         IF $IN[1896] AND NOT $IN[2172] AND $IN[2171] AND $OUT[4039] OR $TIMER_FLAG[8] THEN
            PREVSTEP = $APP_INT[5]
            $APP_INT[5] = 181
         ENDIF
      ;ENDFOLD
   ;ENDFOLD
   ;FOLD SCHRITT 181 --MS2 Reinigung (an Pneum. Schwenkeinheit MS2)-- ;%{P}%MKUKATPVW,%CSTEP,%VST_NR,%P 1:SCHRITT, 2:181, 3:MS2 Reinigung (an Pneum. Schwenkeinheit MS2)
      ;FOLD ;%{H}
         Case 181
      ;ENDFOLD
      ;FOLD -- Steuerluft EIN -- ;%{SE}%MKUKATPVW %CVW_COM %VCOMMENT %P 2:-- Steuerluft EIN --, 3: VW_COMMENT
      ;ENDFOLD
      ;FOLD A2169 = A4039 ;%{SE}%MKUKATPVW %CVW_SPS %VBOASG %P 2:A2169 = A4039, 3: BOASG
         $OUT[2169] = $OUT[4039]
      ;ENDFOLD
      ;FOLD -- RSK Fehlerausgabe Schwenkeinheit 2 Ruhestellung -- ;%{SE}%MKUKATPVW %CVW_COM %VCOMMENT %P 2:-- RSK Fehlerausgabe Schwenkeinheit 2 Ruhestellung --, 3: VW_COMMENT
      ;ENDFOLD
      ;FOLD F323 = !E2171 & T8 + F323 ;%{SE}%MKUKATPVW %CVW_SPS %VBOASG %P 2:F323 = !E2171 & T8 + F323, 3: BOASG
         $FLAG[323] = NOT $IN[2171] AND $TIMER_FLAG[8] OR $FLAG[323]
      ;ENDFOLD
      ;FOLD -- RSK Sammelstoerung -- ;%{SE}%MKUKATPVW %CVW_COM %VCOMMENT %P 2:-- RSK Sammelstoerung --, 3: VW_COMMENT
      ;ENDFOLD
      ;FOLD F329 = F323 ;%{SE}%MKUKATPVW %CVW_SPS %VBOASG %P 2:F329 = F323, 3: BOASG
         $FLAG[329] = $FLAG[323]
      ;ENDFOLD
      ;FOLD A2171 = AUS ;%{SE}%MKUKATPVW %CVW_SPS %VBOASG %P 2:A2171 = AUS, 3: BOASG
         $OUT[2171] = FALSE
      ;ENDFOLD
      ;FOLD -- FRG Bewegung AUS -- ;%{SE}%MKUKATPVW %CVW_COM %VCOMMENT %P 2:-- FRG Bewegung AUS --, 3: VW_COMMENT
      ;ENDFOLD
      ;FOLD A2174 = AUS ;%{SE}%MKUKATPVW %CVW_SPS %VBOASG %P 2:A2174 = AUS, 3: BOASG
         $OUT[2174] = FALSE
      ;ENDFOLD
      ;FOLD Schritt 178 = F323 & (E26 + E27) & A4039 ;%{SE}%MKUKATPVW %CVW_SPS %VST_CON %P 2:Schritt 178 = F323 & (E26 + E27) & A4039, 3: ST_CON
         IF $FLAG[323] AND ($IN[26] OR $IN[27]) AND $OUT[4039] THEN
            PREVSTEP = $APP_INT[5]
            $APP_INT[5] = 178
         ENDIF
      ;ENDFOLD
      ;FOLD Schritt 182 = !F323 & E2174 & A4039 ;%{SE}%MKUKATPVW %CVW_SPS %VST_CON %P 2:Schritt 182 = !F323 & E2174 & A4039, 3: ST_CON
         IF NOT $FLAG[323] AND $IN[2174] AND $OUT[4039] THEN
            PREVSTEP = $APP_INT[5]
            $APP_INT[5] = 182
         ENDIF
      ;ENDFOLD
   ;ENDFOLD
   ;FOLD SCHRITT 182 --MS2 Reinigung (an Pneum. Schwenkeinheit MS2)-- ;%{P}%MKUKATPVW,%CSTEP,%VST_NR,%P 1:SCHRITT, 2:182, 3:MS2 Reinigung (an Pneum. Schwenkeinheit MS2)
      ;FOLD ;%{H}
         Case 182
      ;ENDFOLD
      ;FOLD -- Steuerluft EIN -- ;%{SE}%MKUKATPVW %CVW_COM %VCOMMENT %P 2:-- Steuerluft EIN --, 3: VW_COMMENT
      ;ENDFOLD
      ;FOLD A2169 = A4039 ;%{SE}%MKUKATPVW %CVW_SPS %VBOASG %P 2:A2169 = A4039, 3: BOASG
         $OUT[2169] = $OUT[4039]
      ;ENDFOLD
      ;FOLD F329 = T8 ;%{SE}%MKUKATPVW %CVW_SPS %VBOASG %P 2:F329 = T8, 3: BOASG
         $FLAG[329] = $TIMER_FLAG[8]
      ;ENDFOLD
      ;FOLD F323 = AUS ;%{SE}%MKUKATPVW %CVW_SPS %VBOASG %P 2:F323 = AUS, 3: BOASG
         $FLAG[323] = FALSE
      ;ENDFOLD
      ;FOLD -- FRG in Endlage halten ein -- ;%{SE}%MKUKATPVW %CVW_COM %VCOMMENT %P 2:-- FRG in Endlage halten ein --, 3: VW_COMMENT
      ;ENDFOLD
      ;FOLD A2173 = EIN ;%{SE}%MKUKATPVW %CVW_SPS %VBOASG %P 2:A2173 = EIN, 3: BOASG
         $OUT[2173] = TRUE
      ;ENDFOLD
      ;FOLD Schritt 183 = E2173 & A4039 ;%{SE}%MKUKATPVW %CVW_SPS %VST_CON %P 2:Schritt 183 = E2173 & A4039, 3: ST_CON
         IF $IN[2173] AND $OUT[4039] THEN
            PREVSTEP = $APP_INT[5]
            $APP_INT[5] = 183
         ENDIF
      ;ENDFOLD
   ;ENDFOLD
   ;FOLD SCHRITT 183 --MS2 Reinigung (an Pneum. Schwenkeinheit MS2)-- ;%{P}%MKUKATPVW,%CSTEP,%VST_NR,%P 1:SCHRITT, 2:183, 3:MS2 Reinigung (an Pneum. Schwenkeinheit MS2)
      ;FOLD ;%{H}
         Case 183
      ;ENDFOLD
      ;FOLD -- Steuerluft EIN -- ;%{SE}%MKUKATPVW %CVW_COM %VCOMMENT %P 2:-- Steuerluft EIN --, 3: VW_COMMENT
      ;ENDFOLD
      ;FOLD A2169 = A4039 ;%{SE}%MKUKATPVW %CVW_SPS %VBOASG %P 2:A2169 = A4039, 3: BOASG
         $OUT[2169] = $OUT[4039]
      ;ENDFOLD
      ;FOLD -- FRG in Endlage halten AUS -- ;%{SE}%MKUKATPVW %CVW_COM %VCOMMENT %P 2:-- FRG in Endlage halten AUS --, 3: VW_COMMENT
      ;ENDFOLD
      ;FOLD A2173 = AUS ;%{SE}%MKUKATPVW %CVW_SPS %VBOASG %P 2:A2173 = AUS, 3: BOASG
         $OUT[2173] = FALSE
      ;ENDFOLD
      ;FOLD -- MS1 Zaehler ruecksetzen -- ;%{SE}%MKUKATPVW %CVW_COM %VCOMMENT %P 2:-- MS1 Zaehler ruecksetzen --, 3: VW_COMMENT
      ;ENDFOLD
      ;FOLD -- MS1 FRG Reinigung -- ;%{SE}%MKUKATPVW %CVW_COM %VCOMMENT %P 2:-- MS1 FRG Reinigung --, 3: VW_COMMENT
      ;ENDFOLD
      ;FOLD F607 = AUS ;%{SE}%MKUKATPVW %CVW_SPS %VBOASG %P 2:F607 = AUS, 3: BOASG
         $FLAG[607] = FALSE
      ;ENDFOLD
      ;FOLD -- MS1 Reinigung FK -- ;%{SE}%MKUKATPVW %CVW_COM %VCOMMENT %P 2:-- MS1 Reinigung FK --, 3: VW_COMMENT
      ;ENDFOLD
      ;FOLD F609 = EIN ;%{SE}%MKUKATPVW %CVW_SPS %VBOASG %P 2:F609 = EIN, 3: BOASG
         $FLAG[609] = TRUE
      ;ENDFOLD
      ;FOLD t8 ( EIN ) = STOP ;%{SE}%MKUKATPVW %CVW_SPS %VTSTOP %P 2:t8 ( EIN ) = STOP, 3: TSTOP
         VW(#SET_TIME,TRUE,8,1,0)
      ;ENDFOLD
      ;FOLD Schritt 1 = A4039 ;%{SE}%MKUKATPVW %CVW_SPS %VST_CON %P 2:Schritt 1 = A4039, 3: ST_CON
         IF $OUT[4039] THEN
            PREVSTEP = $APP_INT[5]
            $APP_INT[5] = 1
         ENDIF
      ;ENDFOLD
   ;ENDFOLD
   ;FOLD SCHRITT 184 -- Reserviert -- ;%{P}%MKUKATPVW,%CSTEP,%VST_NR,%P 1:SCHRITT, 2:184, 3: Reserviert
      ;FOLD ;%{H}
         Case 184
      ;ENDFOLD
      ;FOLD 1:;%{SE} %MKUKATPVW
      ;ENDFOLD
   ;ENDFOLD
   ;FOLD SCHRITT 185 -- Reserviert -- ;%{P}%MKUKATPVW,%CSTEP,%VST_NR,%P 1:SCHRITT, 2:185, 3: Reserviert
      ;FOLD ;%{H}
         Case 185
      ;ENDFOLD
      ;FOLD 1:;%{SE} %MKUKATPVW
      ;ENDFOLD
   ;ENDFOLD
   ;FOLD SCHRITT 186 -- Reserviert -- ;%{P}%MKUKATPVW,%CSTEP,%VST_NR,%P 1:SCHRITT, 2:186, 3: Reserviert
      ;FOLD ;%{H}
         Case 186
      ;ENDFOLD
      ;FOLD 1:;%{SE} %MKUKATPVW
      ;ENDFOLD
   ;ENDFOLD
   ;FOLD SCHRITT 187 -- Reserviert -- ;%{P}%MKUKATPVW,%CSTEP,%VST_NR,%P 1:SCHRITT, 2:187, 3: Reserviert
      ;FOLD ;%{H}
         Case 187
      ;ENDFOLD
      ;FOLD 1:;%{SE} %MKUKATPVW
      ;ENDFOLD
   ;ENDFOLD
   ;FOLD SCHRITT 188 -- Reserviert -- ;%{P}%MKUKATPVW,%CSTEP,%VST_NR,%P 1:SCHRITT, 2:188, 3: Reserviert
      ;FOLD ;%{H}
         Case 188
      ;ENDFOLD
      ;FOLD 1:;%{SE} %MKUKATPVW
      ;ENDFOLD
   ;ENDFOLD
   ;FOLD SCHRITT 189 -- Reserviert -- ;%{P}%MKUKATPVW,%CSTEP,%VST_NR,%P 1:SCHRITT, 2:189, 3: Reserviert
      ;FOLD ;%{H}
         Case 189
      ;ENDFOLD
      ;FOLD 1:;%{SE} %MKUKATPVW
      ;ENDFOLD
   ;ENDFOLD
   ;FOLD SCHRITT 190 -- Reserviert -- ;%{P}%MKUKATPVW,%CSTEP,%VST_NR,%P 1:SCHRITT, 2:190, 3: Reserviert
      ;FOLD ;%{H}
         Case 190
      ;ENDFOLD
      ;FOLD 1:;%{SE} %MKUKATPVW
      ;ENDFOLD
   ;ENDFOLD
   ;FOLD SCHRITT 191 -- Reserviert -- ;%{P}%MKUKATPVW,%CSTEP,%VST_NR,%P 1:SCHRITT, 2:191, 3: Reserviert
      ;FOLD ;%{H}
         Case 191
      ;ENDFOLD
      ;FOLD 1:;%{SE} %MKUKATPVW
      ;ENDFOLD
   ;ENDFOLD
   ;FOLD SCHRITT 192 -- Reserviert -- ;%{P}%MKUKATPVW,%CSTEP,%VST_NR,%P 1:SCHRITT, 2:192, 3: Reserviert
      ;FOLD ;%{H}
         Case 192
      ;ENDFOLD
      ;FOLD 1:;%{SE} %MKUKATPVW
      ;ENDFOLD
   ;ENDFOLD
   ;FOLD SCHRITT 193 -- Reserviert -- ;%{P}%MKUKATPVW,%CSTEP,%VST_NR,%P 1:SCHRITT, 2:193, 3: Reserviert
      ;FOLD ;%{H}
         Case 193
      ;ENDFOLD
      ;FOLD 1:;%{SE} %MKUKATPVW
      ;ENDFOLD
   ;ENDFOLD
   ;FOLD SCHRITT 194 -- Reserviert -- ;%{P}%MKUKATPVW,%CSTEP,%VST_NR,%P 1:SCHRITT, 2:194, 3: Reserviert
      ;FOLD ;%{H}
         Case 194
      ;ENDFOLD
      ;FOLD 1:;%{SE} %MKUKATPVW
      ;ENDFOLD
   ;ENDFOLD
   ;FOLD SCHRITT 195 -- Reserviert -- ;%{P}%MKUKATPVW,%CSTEP,%VST_NR,%P 1:SCHRITT, 2:195, 3: Reserviert
      ;FOLD ;%{H}
         Case 195
      ;ENDFOLD
      ;FOLD 1:;%{SE} %MKUKATPVW
      ;ENDFOLD
   ;ENDFOLD
   ;FOLD SCHRITT 196 -- Reserviert -- ;%{P}%MKUKATPVW,%CSTEP,%VST_NR,%P 1:SCHRITT, 2:196, 3: Reserviert
      ;FOLD ;%{H}
         Case 196
      ;ENDFOLD
      ;FOLD 1:;%{SE} %MKUKATPVW
      ;ENDFOLD
   ;ENDFOLD
   ;FOLD SCHRITT 197 -- Reserviert -- ;%{P}%MKUKATPVW,%CSTEP,%VST_NR,%P 1:SCHRITT, 2:197, 3: Reserviert
      ;FOLD ;%{H}
         Case 197
      ;ENDFOLD
      ;FOLD 1:;%{SE} %MKUKATPVW
      ;ENDFOLD
   ;ENDFOLD
   ;FOLD SCHRITT 198 -- Reserviert -- ;%{P}%MKUKATPVW,%CSTEP,%VST_NR,%P 1:SCHRITT, 2:198, 3: Reserviert
      ;FOLD ;%{H}
         Case 198
      ;ENDFOLD
      ;FOLD 1:;%{SE} %MKUKATPVW
      ;ENDFOLD
   ;ENDFOLD
   ;FOLD SCHRITT 199 -- Reserviert -- ;%{P}%MKUKATPVW,%CSTEP,%VST_NR,%P 1:SCHRITT, 2:199, 3: Reserviert
      ;FOLD ;%{H}
         Case 199
      ;ENDFOLD
      ;FOLD 1:;%{SE} %MKUKATPVW
      ;ENDFOLD
   ;ENDFOLD
   ;FOLD SCHRITT 200 -- Reserviert -- ;%{P}%MKUKATPVW,%CSTEP,%VST_NR,%P 1:SCHRITT, 2:200, 3: Reserviert
      ;FOLD ;%{H}
         Case 200
      ;ENDFOLD
      ;FOLD 1:;%{SE} %MKUKATPVW
      ;ENDFOLD
   ;ENDFOLD
   ;FOLD SCHRITT 201 -- Reserviert -- ;%{P}%MKUKATPVW,%CSTEP,%VST_NR,%P 1:SCHRITT, 2:201, 3: Reserviert
      ;FOLD ;%{H}
         Case 201
      ;ENDFOLD
      ;FOLD 1:;%{SE} %MKUKATPVW
      ;ENDFOLD
   ;ENDFOLD
   ;FOLD SCHRITT 202 -- Reserviert -- ;%{P}%MKUKATPVW,%CSTEP,%VST_NR,%P 1:SCHRITT, 2:202, 3: Reserviert
      ;FOLD ;%{H}
         Case 202
      ;ENDFOLD
      ;FOLD 1:;%{SE} %MKUKATPVW
      ;ENDFOLD
   ;ENDFOLD
   ;FOLD SCHRITT 203 -- Reserviert -- ;%{P}%MKUKATPVW,%CSTEP,%VST_NR,%P 1:SCHRITT, 2:203, 3: Reserviert
      ;FOLD ;%{H}
         Case 203
      ;ENDFOLD
      ;FOLD 1:;%{SE} %MKUKATPVW
      ;ENDFOLD
   ;ENDFOLD
   ;FOLD SCHRITT 204 -- Reserviert -- ;%{P}%MKUKATPVW,%CSTEP,%VST_NR,%P 1:SCHRITT, 2:204, 3: Reserviert
      ;FOLD ;%{H}
         Case 204
      ;ENDFOLD
      ;FOLD 1:;%{SE} %MKUKATPVW
      ;ENDFOLD
   ;ENDFOLD
   ;FOLD SCHRITT 205 -- Reserviert -- ;%{P}%MKUKATPVW,%CSTEP,%VST_NR,%P 1:SCHRITT, 2:205, 3: Reserviert
      ;FOLD ;%{H}
         Case 205
      ;ENDFOLD
      ;FOLD 1:;%{SE} %MKUKATPVW
      ;ENDFOLD
   ;ENDFOLD
   ;FOLD SCHRITT 206 -- Reserviert -- ;%{P}%MKUKATPVW,%CSTEP,%VST_NR,%P 1:SCHRITT, 2:206, 3: Reserviert
      ;FOLD ;%{H}
         Case 206
      ;ENDFOLD
      ;FOLD 1:;%{SE} %MKUKATPVW
      ;ENDFOLD
   ;ENDFOLD
   ;FOLD SCHRITT 207 -- Reserviert -- ;%{P}%MKUKATPVW,%CSTEP,%VST_NR,%P 1:SCHRITT, 2:207, 3: Reserviert
      ;FOLD ;%{H}
         Case 207
      ;ENDFOLD
      ;FOLD 1:;%{SE} %MKUKATPVW
      ;ENDFOLD
   ;ENDFOLD
   ;FOLD SCHRITT 208 -- Reserviert -- ;%{P}%MKUKATPVW,%CSTEP,%VST_NR,%P 1:SCHRITT, 2:208, 3: Reserviert
      ;FOLD ;%{H}
         Case 208
      ;ENDFOLD
      ;FOLD 1:;%{SE} %MKUKATPVW
      ;ENDFOLD
   ;ENDFOLD
   ;FOLD SCHRITT 209 -- Reserviert -- ;%{P}%MKUKATPVW,%CSTEP,%VST_NR,%P 1:SCHRITT, 2:209, 3: Reserviert
      ;FOLD ;%{H}
         Case 209
      ;ENDFOLD
      ;FOLD 1:;%{SE} %MKUKATPVW
      ;ENDFOLD
   ;ENDFOLD
   ;FOLD SCHRITT 210 -- Reserviert -- ;%{P}%MKUKATPVW,%CSTEP,%VST_NR,%P 1:SCHRITT, 2:210, 3: Reserviert
      ;FOLD ;%{H}
         Case 210
      ;ENDFOLD
      ;FOLD 1:;%{SE} %MKUKATPVW
      ;ENDFOLD
   ;ENDFOLD
   ;FOLD SCHRITT 211 -- Reserviert -- ;%{P}%MKUKATPVW,%CSTEP,%VST_NR,%P 1:SCHRITT, 2:211, 3: Reserviert
      ;FOLD ;%{H}
         Case 211
      ;ENDFOLD
      ;FOLD 1:;%{SE} %MKUKATPVW
      ;ENDFOLD
   ;ENDFOLD
   ;FOLD SCHRITT 212 -- Reserviert -- ;%{P}%MKUKATPVW,%CSTEP,%VST_NR,%P 1:SCHRITT, 2:212, 3: Reserviert
      ;FOLD ;%{H}
         Case 212
      ;ENDFOLD
      ;FOLD 1:;%{SE} %MKUKATPVW
      ;ENDFOLD
   ;ENDFOLD
   ;FOLD SCHRITT 213 -- Reserviert -- ;%{P}%MKUKATPVW,%CSTEP,%VST_NR,%P 1:SCHRITT, 2:213, 3: Reserviert
      ;FOLD ;%{H}
         Case 213
      ;ENDFOLD
      ;FOLD 1:;%{SE} %MKUKATPVW
      ;ENDFOLD
   ;ENDFOLD
   ;FOLD SCHRITT 214 -- Reserviert -- ;%{P}%MKUKATPVW,%CSTEP,%VST_NR,%P 1:SCHRITT, 2:214, 3: Reserviert
      ;FOLD ;%{H}
         Case 214
      ;ENDFOLD
      ;FOLD 1:;%{SE} %MKUKATPVW
      ;ENDFOLD
   ;ENDFOLD
   ;FOLD SCHRITT 215 -- Reserviert -- ;%{P}%MKUKATPVW,%CSTEP,%VST_NR,%P 1:SCHRITT, 2:215, 3: Reserviert
      ;FOLD ;%{H}
         Case 215
      ;ENDFOLD
      ;FOLD 1:;%{SE} %MKUKATPVW
      ;ENDFOLD
   ;ENDFOLD
   ;FOLD SCHRITT 216 -- Reserviert -- ;%{P}%MKUKATPVW,%CSTEP,%VST_NR,%P 1:SCHRITT, 2:216, 3: Reserviert
      ;FOLD ;%{H}
         Case 216
      ;ENDFOLD
      ;FOLD 1:;%{SE} %MKUKATPVW
      ;ENDFOLD
   ;ENDFOLD
   ;FOLD SCHRITT 217 -- STAT EZ1/SP1/KE1 Setzhub 2 -- ;%{P}%MKUKATPVW,%CSTEP,%VST_NR,%P 1:SCHRITT, 2:217, 3: STAT EZ1/SP1/KE1 Setzhub 2
      ;FOLD ;%{H}
         Case 217
      ;ENDFOLD
      ;FOLD -- Druckvorgabe SK1/EZ1/SP1/KE1 -- ;%{SE}%MKUKATPVW %CVW_COM %VCOMMENT %P 2:-- Druckvorgabe SK1/EZ1/SP1/KE1 --, 3: VW_COMMENT
      ;ENDFOLD
      ;FOLD F168 = F78 & !F830 ;%{SE}%MKUKATPVW %CVW_SPS %VBOASG %P 2:F168 = F78 & !F830, 3: BOASG
         $FLAG[168] = $FLAG[78] AND NOT $FLAG[830]
      ;ENDFOLD
      ;FOLD bin1 ( F168 ) = 61 ;%{SE}%MKUKATPVW %CVW_SPS %VARIASG %P 2:bin1 ( F168 ) = 61, 3: ARIASG
         VW(#BINOUT,$FLAG[168],1,61)
      ;ENDFOLD
      ;FOLD F168 = AUS ;%{SE}%MKUKATPVW %CVW_SPS %VBOASG %P 2:F168 = AUS, 3: BOASG
         $FLAG[168] = FALSE
      ;ENDFOLD
      ;FOLD bin3 ( F78 ) = 61 ;%{SE}%MKUKATPVW %CVW_SPS %VARIASG %P 2:bin3 ( F78 ) = 61, 3: ARIASG
         VW(#BINOUT,$FLAG[78],3,61)
      ;ENDFOLD
      ;FOLD -- Wartezeit Programmwechsel SK -- ;%{SE}%MKUKATPVW %CVW_COM %VCOMMENT %P 2:-- Wartezeit Programmwechsel SK --, 3: VW_COMMENT
      ;ENDFOLD
      ;FOLD T8 ( !F334 ) = -2[1/10Sek] ;%{SE}%MKUKATPVW %CVW_SPS %VTASG %P 2:T8 ( !F334 ) = -2[1/10Sek], 3: TASG
         VW(#SET_TIME,NOT $FLAG[334],8,0,-2)
      ;ENDFOLD
      ;FOLD -- Hilfsflag SK Programmwechsel -- ;%{SE}%MKUKATPVW %CVW_COM %VCOMMENT %P 2:-- Hilfsflag SK Programmwechsel --, 3: VW_COMMENT
      ;ENDFOLD
      ;FOLD F334 = EIN ;%{SE}%MKUKATPVW %CVW_SPS %VBOASG %P 2:F334 = EIN, 3: BOASG
         $FLAG[334] = TRUE
      ;ENDFOLD
      ;FOLD Schritt 218 = T8 & A4039 ;%{SE}%MKUKATPVW %CVW_SPS %VST_CON %P 2:Schritt 218 = T8 & A4039, 3: ST_CON
         IF $TIMER_FLAG[8] AND $OUT[4039] THEN
            PREVSTEP = $APP_INT[5]
            $APP_INT[5] = 218
         ENDIF
      ;ENDFOLD
   ;ENDFOLD
   ;FOLD SCHRITT 218 -- STAT EZ1/SP1/KE1 Setzhub 2 -- ;%{P}%MKUKATPVW,%CSTEP,%VST_NR,%P 1:SCHRITT, 2:218, 3: STAT EZ1/SP1/KE1 Setzhub 2
      ;FOLD ;%{H}
         Case 218
      ;ENDFOLD
      ;FOLD -- Hilfsflag SK Programmwechsel -- ;%{SE}%MKUKATPVW %CVW_COM %VCOMMENT %P 2:-- Hilfsflag SK Programmwechsel --, 3: VW_COMMENT
      ;ENDFOLD
      ;FOLD F334 = AUS ;%{SE}%MKUKATPVW %CVW_SPS %VBOASG %P 2:F334 = AUS, 3: BOASG
         $FLAG[334] = FALSE
      ;ENDFOLD
      ;FOLD -- Zeit fuer Setzhub -- ;%{SE}%MKUKATPVW %CVW_COM %VCOMMENT %P 2:-- Zeit fuer Setzhub --, 3: VW_COMMENT
      ;ENDFOLD
      ;FOLD T8 ( EIN ) = -15[1/10Sek] ;%{SE}%MKUKATPVW %CVW_SPS %VTASG %P 2:T8 ( EIN ) = -15[1/10Sek], 3: TASG
         VW(#SET_TIME,TRUE,8,0,-15)
      ;ENDFOLD
      ;FOLD Schritt 219 = A4039 ;%{SE}%MKUKATPVW %CVW_SPS %VST_CON %P 2:Schritt 219 = A4039, 3: ST_CON
         IF $OUT[4039] THEN
            PREVSTEP = $APP_INT[5]
            $APP_INT[5] = 219
         ENDIF
      ;ENDFOLD
   ;ENDFOLD
   ;FOLD SCHRITT 219 -- STAT EZ1/SP1/KE1 Setzhub 2 -- ;%{P}%MKUKATPVW,%CSTEP,%VST_NR,%P 1:SCHRITT, 2:219, 3: STAT EZ1/SP1/KE1 Setzhub 2
      ;FOLD ;%{H}
         Case 219
      ;ENDFOLD
      ;FOLD -- Hilfsflag SK Programmwechsel -- ;%{SE}%MKUKATPVW %CVW_COM %VCOMMENT %P 2:-- Hilfsflag SK Programmwechsel --, 3: VW_COMMENT
      ;ENDFOLD
      ;FOLD F334 = AUS ;%{SE}%MKUKATPVW %CVW_SPS %VBOASG %P 2:F334 = AUS, 3: BOASG
         $FLAG[334] = FALSE
      ;ENDFOLD
      ;FOLD -- EZ1/SP1/KE1 schliessen -- ;%{SE}%MKUKATPVW %CVW_COM %VCOMMENT %P 2:-- EZ1/SP1/KE1 schliessen --, 3: VW_COMMENT
      ;ENDFOLD
      ;FOLD A717 = AUS ;%{SE}%MKUKATPVW %CVW_SPS %VBOASG %P 2:A717 = AUS, 3: BOASG
         $OUT[717] = FALSE
      ;ENDFOLD
      ;FOLD -- EZ1/SP1 -- ;%{SE}%MKUKATPVW %CVW_COM %VCOMMENT %P 2:-- EZ1/SP1 --, 3: VW_COMMENT
      ;ENDFOLD
      ;FOLD A718 = !F329 & !F122 & !F830 ;%{SE}%MKUKATPVW %CVW_SPS %VBOASG %P 2:A718 = !F329 & !F122 & !F830, 3: BOASG
         $OUT[718] = NOT $FLAG[329] AND NOT $FLAG[122] AND NOT $FLAG[830]
      ;ENDFOLD
      ;FOLD -- KE1 -- ;%{SE}%MKUKATPVW %CVW_COM %VCOMMENT %P 2:-- KE1 --, 3: VW_COMMENT
      ;ENDFOLD
      ;FOLD A766 = !F329 & !F122 & F830 ;%{SE}%MKUKATPVW %CVW_SPS %VBOASG %P 2:A766 = !F329 & !F122 & F830, 3: BOASG
         $OUT[766] = NOT $FLAG[329] AND NOT $FLAG[122] AND $FLAG[830]
      ;ENDFOLD
      ;FOLD Schritt 220 = (!E717 & E718 & T8 + T9) & A4039 ;%{SE}%MKUKATPVW %CVW_SPS %VST_CON %P 2:Schritt 220 = (!E717 & E718 & T8 + T9) & A4039, 3: ST_CON
         IF (NOT $IN[717] AND $IN[718] AND $TIMER_FLAG[8] OR $TIMER_FLAG[9]) AND $OUT[4039] THEN
            PREVSTEP = $APP_INT[5]
            $APP_INT[5] = 220
         ENDIF
      ;ENDFOLD
   ;ENDFOLD
   ;FOLD SCHRITT 220 -- STAT EZ1/SP1/KE1 Setzhub 2 -- ;%{P}%MKUKATPVW,%CSTEP,%VST_NR,%P 1:SCHRITT, 2:220, 3: STAT EZ1/SP1/KE1 Setzhub 2
      ;FOLD ;%{H}
         Case 220
      ;ENDFOLD
      ;FOLD -- RSK Fehlerausgabe Kraftaufbau -- ;%{SE}%MKUKATPVW %CVW_COM %VCOMMENT %P 2:-- RSK Fehlerausgabe Kraftaufbau --, 3: VW_COMMENT
      ;ENDFOLD
      ;FOLD F325 = !E718 & T9 ;%{SE}%MKUKATPVW %CVW_SPS %VBOASG %P 2:F325 = !E718 & T9, 3: BOASG
         $FLAG[325] = NOT $IN[718] AND $TIMER_FLAG[9]
      ;ENDFOLD
      ;FOLD F329 = T9 ;%{SE}%MKUKATPVW %CVW_SPS %VBOASG %P 2:F329 = T9, 3: BOASG
         $FLAG[329] = $TIMER_FLAG[9]
      ;ENDFOLD
      ;FOLD -- EZ1/SP1/KE1 SZ1 oeffnen -- ;%{SE}%MKUKATPVW %CVW_COM %VCOMMENT %P 2:-- EZ1/SP1/KE1 SZ1 oeffnen --, 3: VW_COMMENT
      ;ENDFOLD
      ;FOLD A718 = AUS ;%{SE}%MKUKATPVW %CVW_SPS %VBOASG %P 2:A718 = AUS, 3: BOASG
         $OUT[718] = FALSE
      ;ENDFOLD
      ;FOLD A766 = AUS ;%{SE}%MKUKATPVW %CVW_SPS %VBOASG %P 2:A766 = AUS, 3: BOASG
         $OUT[766] = FALSE
      ;ENDFOLD
      ;FOLD A717 = EIN ;%{SE}%MKUKATPVW %CVW_SPS %VBOASG %P 2:A717 = EIN, 3: BOASG
         $OUT[717] = TRUE
      ;ENDFOLD
      ;FOLD -- Druckvorgabe SK1/EZ1/SP1/KE1 -- ;%{SE}%MKUKATPVW %CVW_COM %VCOMMENT %P 2:-- Druckvorgabe SK1/EZ1/SP1/KE1 --, 3: VW_COMMENT
      ;ENDFOLD
      ;FOLD F168 = F78 & !F830 ;%{SE}%MKUKATPVW %CVW_SPS %VBOASG %P 2:F168 = F78 & !F830, 3: BOASG
         $FLAG[168] = $FLAG[78] AND NOT $FLAG[830]
      ;ENDFOLD
      ;FOLD bin1 ( F168 ) = 41 ;%{SE}%MKUKATPVW %CVW_SPS %VARIASG %P 2:bin1 ( F168 ) = 41, 3: ARIASG
         VW(#BINOUT,$FLAG[168],1,41)
      ;ENDFOLD
      ;FOLD F168 = F79 & !F830 ;%{SE}%MKUKATPVW %CVW_SPS %VBOASG %P 2:F168 = F79 & !F830, 3: BOASG
         $FLAG[168] = $FLAG[79] AND NOT $FLAG[830]
      ;ENDFOLD
      ;FOLD bin1 ( F79 ) = 51 ;%{SE}%MKUKATPVW %CVW_SPS %VARIASG %P 2:bin1 ( F79 ) = 51, 3: ARIASG
         VW(#BINOUT,$FLAG[79],1,51)
      ;ENDFOLD
      ;FOLD F168 = AUS ;%{SE}%MKUKATPVW %CVW_SPS %VBOASG %P 2:F168 = AUS, 3: BOASG
         $FLAG[168] = FALSE
      ;ENDFOLD
      ;FOLD bin3 ( F78 ) = 41 ;%{SE}%MKUKATPVW %CVW_SPS %VARIASG %P 2:bin3 ( F78 ) = 41, 3: ARIASG
         VW(#BINOUT,$FLAG[78],3,41)
      ;ENDFOLD
      ;FOLD bin3 ( F79 ) = 51 ;%{SE}%MKUKATPVW %CVW_SPS %VARIASG %P 2:bin3 ( F79 ) = 51, 3: ARIASG
         VW(#BINOUT,$FLAG[79],3,51)
      ;ENDFOLD
      ;FOLD -- Wartezeit Programmwechsel SK -- ;%{SE}%MKUKATPVW %CVW_COM %VCOMMENT %P 2:-- Wartezeit Programmwechsel SK --, 3: VW_COMMENT
      ;ENDFOLD
      ;FOLD T8 ( !F334 ) = -2[1/10Sek] ;%{SE}%MKUKATPVW %CVW_SPS %VTASG %P 2:T8 ( !F334 ) = -2[1/10Sek], 3: TASG
         VW(#SET_TIME,NOT $FLAG[334],8,0,-2)
      ;ENDFOLD
      ;FOLD -- Hilfsflag SK Programmwechsel -- ;%{SE}%MKUKATPVW %CVW_COM %VCOMMENT %P 2:-- Hilfsflag SK Programmwechsel --, 3: VW_COMMENT
      ;ENDFOLD
      ;FOLD F334 = EIN ;%{SE}%MKUKATPVW %CVW_SPS %VBOASG %P 2:F334 = EIN, 3: BOASG
         $FLAG[334] = TRUE
      ;ENDFOLD
      ;FOLD Schritt 221 = T8 & A4039 ;%{SE}%MKUKATPVW %CVW_SPS %VST_CON %P 2:Schritt 221 = T8 & A4039, 3: ST_CON
         IF $TIMER_FLAG[8] AND $OUT[4039] THEN
            PREVSTEP = $APP_INT[5]
            $APP_INT[5] = 221
         ENDIF
      ;ENDFOLD
   ;ENDFOLD
   ;FOLD SCHRITT 221 -- STAT EZ1/SP1/KE1 Setzhub 2 -- ;%{P}%MKUKATPVW,%CSTEP,%VST_NR,%P 1:SCHRITT, 2:221, 3: STAT EZ1/SP1/KE1 Setzhub 2
      ;FOLD ;%{H}
         Case 221
      ;ENDFOLD
      ;FOLD -- Hilfsflag SK Programmwechsel -- ;%{SE}%MKUKATPVW %CVW_COM %VCOMMENT %P 2:-- Hilfsflag SK Programmwechsel --, 3: VW_COMMENT
      ;ENDFOLD
      ;FOLD F334 = AUS ;%{SE}%MKUKATPVW %CVW_SPS %VBOASG %P 2:F334 = AUS, 3: BOASG
         $FLAG[334] = FALSE
      ;ENDFOLD
      ;FOLD Schritt 70 = E717 & !E718 & A4039 ;%{SE}%MKUKATPVW %CVW_SPS %VST_CON %P 2:Schritt 70 = E717 & !E718 & A4039, 3: ST_CON
         IF $IN[717] AND NOT $IN[718] AND $OUT[4039] THEN
            PREVSTEP = $APP_INT[5]
            $APP_INT[5] = 70
         ENDIF
      ;ENDFOLD
   ;ENDFOLD
   ;FOLD SCHRITT 222 -- STAT EZ2/SP2/KE2 Setzhub 2 -- ;%{P}%MKUKATPVW,%CSTEP,%VST_NR,%P 1:SCHRITT, 2:222, 3: STAT EZ2/SP2/KE2 Setzhub 2
      ;FOLD ;%{H}
         Case 222
      ;ENDFOLD
      ;FOLD -- Druckvorgabe SK2/SK1/EZ2/SP2/KE2 -- ;%{SE}%MKUKATPVW %CVW_COM %VCOMMENT %P 2:-- Druckvorgabe SK2/SK1/EZ2/SP2/KE2 --, 3: VW_COMMENT
      ;ENDFOLD
      ;FOLD bin3 (F307) = 65 ;%{SE}%MKUKATPVW %CVW_SPS %VARIASG %P 2:bin3 (F307) = 65, 3: ARIASG
         VW(#BINOUT,$FLAG[307],3,65)
      ;ENDFOLD
      ;FOLD F168 = F138 & !F831 ;%{SE}%MKUKATPVW %CVW_SPS %VBOASG %P 2:F168 = F138 & !F831, 3: BOASG
         $FLAG[168] = $FLAG[138] AND NOT $FLAG[831]
      ;ENDFOLD
      ;FOLD bin4 ( F138 ) = 61 ;%{SE}%MKUKATPVW %CVW_SPS %VARIASG %P 2:bin4 ( F138 ) = 61, 3: ARIASG
         VW(#BINOUT,$FLAG[138],4,61)
      ;ENDFOLD
      ;FOLD F168 = AUS ;%{SE}%MKUKATPVW %CVW_SPS %VBOASG %P 2:F168 = AUS, 3: BOASG
         $FLAG[168] = FALSE
      ;ENDFOLD
      ;FOLD bin6 (F138) = 61 ;%{SE}%MKUKATPVW %CVW_SPS %VARIASG %P 2:bin6 (F138) = 61, 3: ARIASG
         VW(#BINOUT,$FLAG[138],6,61)
      ;ENDFOLD
      ;FOLD -- Wartezeit Programmwechsel SK -- ;%{SE}%MKUKATPVW %CVW_COM %VCOMMENT %P 2:-- Wartezeit Programmwechsel SK --, 3: VW_COMMENT
      ;ENDFOLD
      ;FOLD T8 ( !F334 ) = -2[1/10Sek] ;%{SE}%MKUKATPVW %CVW_SPS %VTASG %P 2:T8 ( !F334 ) = -2[1/10Sek], 3: TASG
         VW(#SET_TIME,NOT $FLAG[334],8,0,-2)
      ;ENDFOLD
      ;FOLD -- Hilfsflag SK Programmwechsel -- ;%{SE}%MKUKATPVW %CVW_COM %VCOMMENT %P 2:-- Hilfsflag SK Programmwechsel --, 3: VW_COMMENT
      ;ENDFOLD
      ;FOLD F334 = EIN ;%{SE}%MKUKATPVW %CVW_SPS %VBOASG %P 2:F334 = EIN, 3: BOASG
         $FLAG[334] = TRUE
      ;ENDFOLD
      ;FOLD Schritt 223 = T8 & A4039 ;%{SE}%MKUKATPVW %CVW_SPS %VST_CON %P 2:Schritt 223 = T8 & A4039, 3: ST_CON
         IF $TIMER_FLAG[8] AND $OUT[4039] THEN
            PREVSTEP = $APP_INT[5]
            $APP_INT[5] = 223
         ENDIF
      ;ENDFOLD
   ;ENDFOLD
   ;FOLD SCHRITT 223 -- STAT EZ1/SP1/KE1 Setzhub 2 -- ;%{P}%MKUKATPVW,%CSTEP,%VST_NR,%P 1:SCHRITT, 2:223, 3: STAT EZ1/SP1/KE1 Setzhub 2
      ;FOLD ;%{H}
         Case 223
      ;ENDFOLD
      ;FOLD -- Hilfsflag SK Programmwechsel -- ;%{SE}%MKUKATPVW %CVW_COM %VCOMMENT %P 2:-- Hilfsflag SK Programmwechsel --, 3: VW_COMMENT
      ;ENDFOLD
      ;FOLD F334 = AUS ;%{SE}%MKUKATPVW %CVW_SPS %VBOASG %P 2:F334 = AUS, 3: BOASG
         $FLAG[334] = FALSE
      ;ENDFOLD
      ;FOLD -- Zeit fuer Setzhub -- ;%{SE}%MKUKATPVW %CVW_COM %VCOMMENT %P 2:-- Zeit fuer Setzhub --, 3: VW_COMMENT
      ;ENDFOLD
      ;FOLD T8 ( EIN ) = -15[1/10Sek] ;%{SE}%MKUKATPVW %CVW_SPS %VTASG %P 2:T8 ( EIN ) = -15[1/10Sek], 3: TASG
         VW(#SET_TIME,TRUE,8,0,-15)
      ;ENDFOLD
      ;FOLD Schritt 224 = A4039 ;%{SE}%MKUKATPVW %CVW_SPS %VST_CON %P 2:Schritt 224 = A4039, 3: ST_CON
         IF $OUT[4039] THEN
            PREVSTEP = $APP_INT[5]
            $APP_INT[5] = 224
         ENDIF
      ;ENDFOLD
   ;ENDFOLD
   ;FOLD SCHRITT 224 -- STAT EZ2/SP2/KE2 Setzhub 2 -- ;%{P}%MKUKATPVW,%CSTEP,%VST_NR,%P 1:SCHRITT, 2:224, 3: STAT EZ2/SP2/KE2 Setzhub 2
      ;FOLD ;%{H}
         Case 224
      ;ENDFOLD
      ;FOLD -- EZ2/SP2/KE2 schliessen -- ;%{SE}%MKUKATPVW %CVW_COM %VCOMMENT %P 2:-- EZ2/SP2/KE2 schliessen --, 3: VW_COMMENT
      ;ENDFOLD
      ;FOLD A877 = AUS ;%{SE}%MKUKATPVW %CVW_SPS %VBOASG %P 2:A877 = AUS, 3: BOASG
         $OUT[877] = FALSE
      ;ENDFOLD
      ;FOLD -- EZ2/SP2 -- ;%{SE}%MKUKATPVW %CVW_COM %VCOMMENT %P 2:-- EZ2/SP2 --, 3: VW_COMMENT
      ;ENDFOLD
      ;FOLD A878 = !F329 & !F160 & !F831 ;%{SE}%MKUKATPVW %CVW_SPS %VBOASG %P 2:A878 = !F329 & !F160 & !F831, 3: BOASG
         $OUT[878] = NOT $FLAG[329] AND NOT $FLAG[160] AND NOT $FLAG[831]
      ;ENDFOLD
      ;FOLD -- KE2 -- ;%{SE}%MKUKATPVW %CVW_COM %VCOMMENT %P 2:-- KE2 --, 3: VW_COMMENT
      ;ENDFOLD
      ;FOLD A926 = !F329 & !F160 & F831 ;%{SE}%MKUKATPVW %CVW_SPS %VBOASG %P 2:A926 = !F329 & !F160 & F831, 3: BOASG
         $OUT[926] = NOT $FLAG[329] AND NOT $FLAG[160] AND $FLAG[831]
      ;ENDFOLD
      ;FOLD Schritt 225 = (!E877 & E878 & T8 + T9) & A4039 ;%{SE}%MKUKATPVW %CVW_SPS %VST_CON %P 2:Schritt 225 = (!E877 & E878 & T8 + T9) & A4039, 3: ST_CON
         IF (NOT $IN[877] AND $IN[878] AND $TIMER_FLAG[8] OR $TIMER_FLAG[9]) AND $OUT[4039] THEN
            PREVSTEP = $APP_INT[5]
            $APP_INT[5] = 225
         ENDIF
      ;ENDFOLD
   ;ENDFOLD
   ;FOLD SCHRITT 225 -- STAT EZ2/SP2/KE2 Setzhub 2 -- ;%{P}%MKUKATPVW,%CSTEP,%VST_NR,%P 1:SCHRITT, 2:225, 3: STAT EZ2/SP2/KE2 Setzhub 2
      ;FOLD ;%{H}
         Case 225
      ;ENDFOLD
      ;FOLD -- RSK Fehlerausgabe Kraftaufbau -- ;%{SE}%MKUKATPVW %CVW_COM %VCOMMENT %P 2:-- RSK Fehlerausgabe Kraftaufbau --, 3: VW_COMMENT
      ;ENDFOLD
      ;FOLD F325 = !E878 & T9 ;%{SE}%MKUKATPVW %CVW_SPS %VBOASG %P 2:F325 = !E878 & T9, 3: BOASG
         $FLAG[325] = NOT $IN[878] AND $TIMER_FLAG[9]
      ;ENDFOLD
      ;FOLD F329 = T9 ;%{SE}%MKUKATPVW %CVW_SPS %VBOASG %P 2:F329 = T9, 3: BOASG
         $FLAG[329] = $TIMER_FLAG[9]
      ;ENDFOLD
      ;FOLD -- EZ2/SP2/KE2 SZ1 oeffnen -- ;%{SE}%MKUKATPVW %CVW_COM %VCOMMENT %P 2:-- EZ2/SP2/KE2 SZ1 oeffnen --, 3: VW_COMMENT
      ;ENDFOLD
      ;FOLD A878 = AUS ;%{SE}%MKUKATPVW %CVW_SPS %VBOASG %P 2:A878 = AUS, 3: BOASG
         $OUT[878] = FALSE
      ;ENDFOLD
      ;FOLD A926 = AUS ;%{SE}%MKUKATPVW %CVW_SPS %VBOASG %P 2:A926 = AUS, 3: BOASG
         $OUT[926] = FALSE
      ;ENDFOLD
      ;FOLD A877 = EIN ;%{SE}%MKUKATPVW %CVW_SPS %VBOASG %P 2:A877 = EIN, 3: BOASG
         $OUT[877] = TRUE
      ;ENDFOLD
      ;FOLD -- Druckvorgabe SK2/SK1/EZ2/SP2/KE2 -- ;%{SE}%MKUKATPVW %CVW_COM %VCOMMENT %P 2:-- Druckvorgabe SK2/SK1/EZ2/SP2/KE2 --, 3: VW_COMMENT
      ;ENDFOLD
      ;FOLD bin3 (F307) = 45 ;%{SE}%MKUKATPVW %CVW_SPS %VARIASG %P 2:bin3 (F307) = 45, 3: ARIASG
         VW(#BINOUT,$FLAG[307],3,45)
      ;ENDFOLD
      ;FOLD bin3 (F308) = 55 ;%{SE}%MKUKATPVW %CVW_SPS %VARIASG %P 2:bin3 (F308) = 55, 3: ARIASG
         VW(#BINOUT,$FLAG[308],3,55)
      ;ENDFOLD
      ;FOLD F168 = F138 & !F831 ;%{SE}%MKUKATPVW %CVW_SPS %VBOASG %P 2:F168 = F138 & !F831, 3: BOASG
         $FLAG[168] = $FLAG[138] AND NOT $FLAG[831]
      ;ENDFOLD
      ;FOLD bin4 (F168) = 41 ;%{SE}%MKUKATPVW %CVW_SPS %VARIASG %P 2:bin4 (F168) = 41, 3: ARIASG
         VW(#BINOUT,$FLAG[168],4,41)
      ;ENDFOLD
      ;FOLD F168 = F139 & !F831 ;%{SE}%MKUKATPVW %CVW_SPS %VBOASG %P 2:F168 = F139 & !F831, 3: BOASG
         $FLAG[168] = $FLAG[139] AND NOT $FLAG[831]
      ;ENDFOLD
      ;FOLD bin4 (F168) = 51 ;%{SE}%MKUKATPVW %CVW_SPS %VARIASG %P 2:bin4 (F168) = 51, 3: ARIASG
         VW(#BINOUT,$FLAG[168],4,51)
      ;ENDFOLD
      ;FOLD F168 = AUS ;%{SE}%MKUKATPVW %CVW_SPS %VBOASG %P 2:F168 = AUS, 3: BOASG
         $FLAG[168] = FALSE
      ;ENDFOLD
      ;FOLD bin6 (F138) = 41 ;%{SE}%MKUKATPVW %CVW_SPS %VARIASG %P 2:bin6 (F138) = 41, 3: ARIASG
         VW(#BINOUT,$FLAG[138],6,41)
      ;ENDFOLD
      ;FOLD bin6 (F139) = 51 ;%{SE}%MKUKATPVW %CVW_SPS %VARIASG %P 2:bin6 (F139) = 51, 3: ARIASG
         VW(#BINOUT,$FLAG[139],6,51)
      ;ENDFOLD
      ;FOLD -- Wartezeit Programmwechsel SK -- ;%{SE}%MKUKATPVW %CVW_COM %VCOMMENT %P 2:-- Wartezeit Programmwechsel SK --, 3: VW_COMMENT
      ;ENDFOLD
      ;FOLD T8 ( !F334 ) = -2[1/10Sek] ;%{SE}%MKUKATPVW %CVW_SPS %VTASG %P 2:T8 ( !F334 ) = -2[1/10Sek], 3: TASG
         VW(#SET_TIME,NOT $FLAG[334],8,0,-2)
      ;ENDFOLD
      ;FOLD -- Hilfsflag SK Programmwechsel -- ;%{SE}%MKUKATPVW %CVW_COM %VCOMMENT %P 2:-- Hilfsflag SK Programmwechsel --, 3: VW_COMMENT
      ;ENDFOLD
      ;FOLD F334 = EIN ;%{SE}%MKUKATPVW %CVW_SPS %VBOASG %P 2:F334 = EIN, 3: BOASG
         $FLAG[334] = TRUE
      ;ENDFOLD
      ;FOLD Schritt 226 = T8 & A4039 ;%{SE}%MKUKATPVW %CVW_SPS %VST_CON %P 2:Schritt 226 = T8 & A4039, 3: ST_CON
         IF $TIMER_FLAG[8] AND $OUT[4039] THEN
            PREVSTEP = $APP_INT[5]
            $APP_INT[5] = 226
         ENDIF
      ;ENDFOLD
   ;ENDFOLD
   ;FOLD SCHRITT 226 -- STAT EZ2/SP2/KE2 Setzhub 2 -- ;%{P}%MKUKATPVW,%CSTEP,%VST_NR,%P 1:SCHRITT, 2:226, 3: STAT EZ2/SP2/KE2 Setzhub 2
      ;FOLD ;%{H}
         Case 226
      ;ENDFOLD
      ;FOLD -- Hilfsflag SK Programmwechsel -- ;%{SE}%MKUKATPVW %CVW_COM %VCOMMENT %P 2:-- Hilfsflag SK Programmwechsel --, 3: VW_COMMENT
      ;ENDFOLD
      ;FOLD F334 = AUS ;%{SE}%MKUKATPVW %CVW_SPS %VBOASG %P 2:F334 = AUS, 3: BOASG
         $FLAG[334] = FALSE
      ;ENDFOLD
      ;FOLD Schritt 93 = E877 & !E878 & A4039 ;%{SE}%MKUKATPVW %CVW_SPS %VST_CON %P 2:Schritt 93 = E877 & !E878 & A4039, 3: ST_CON
         IF $IN[877] AND NOT $IN[878] AND $OUT[4039] THEN
            PREVSTEP = $APP_INT[5]
            $APP_INT[5] = 93
         ENDIF
      ;ENDFOLD
   ;ENDFOLD
   ;FOLD SCHRITT 227 -- STAT EZ3/SP3/KE3 Setzhub 2 -- ;%{P}%MKUKATPVW,%CSTEP,%VST_NR,%P 1:SCHRITT, 2:227, 3: STAT EZ3/SP3/KE3 Setzhub 2
      ;FOLD ;%{H}
         Case 227
      ;ENDFOLD
      ;FOLD -- Druckvorgabe SK3/EZ3/SP3/KE3 -- ;%{SE}%MKUKATPVW %CVW_COM %VCOMMENT %P 2:-- Druckvorgabe SK3/EZ3/SP3/KE3 --, 3: VW_COMMENT
      ;ENDFOLD
      ;FOLD F168 = F174 & !F832 ;%{SE}%MKUKATPVW %CVW_SPS %VBOASG %P 2:F168 = F174 & !F832, 3: BOASG
         $FLAG[168] = $FLAG[174] AND NOT $FLAG[832]
      ;ENDFOLD
      ;FOLD bin7 ( F174 ) = 61 ;%{SE}%MKUKATPVW %CVW_SPS %VARIASG %P 2:bin7 ( F174 ) = 61, 3: ARIASG
         VW(#BINOUT,$FLAG[174],7,61)
      ;ENDFOLD
      ;FOLD F168 = AUS ;%{SE}%MKUKATPVW %CVW_SPS %VBOASG %P 2:F168 = AUS, 3: BOASG
         $FLAG[168] = FALSE
      ;ENDFOLD
      ;FOLD bin9 ( F174 ) = 61 ;%{SE}%MKUKATPVW %CVW_SPS %VARIASG %P 2:bin9 ( F174 ) = 61, 3: ARIASG
         VW(#BINOUT,$FLAG[174],9,61)
      ;ENDFOLD
      ;FOLD -- Wartezeit Programmwechsel SK -- ;%{SE}%MKUKATPVW %CVW_COM %VCOMMENT %P 2:-- Wartezeit Programmwechsel SK --, 3: VW_COMMENT
      ;ENDFOLD
      ;FOLD T8 ( !F334 ) = -2[1/10Sek] ;%{SE}%MKUKATPVW %CVW_SPS %VTASG %P 2:T8 ( !F334 ) = -2[1/10Sek], 3: TASG
         VW(#SET_TIME,NOT $FLAG[334],8,0,-2)
      ;ENDFOLD
      ;FOLD -- Hilfsflag SK Programmwechsel -- ;%{SE}%MKUKATPVW %CVW_COM %VCOMMENT %P 2:-- Hilfsflag SK Programmwechsel --, 3: VW_COMMENT
      ;ENDFOLD
      ;FOLD F334 = EIN ;%{SE}%MKUKATPVW %CVW_SPS %VBOASG %P 2:F334 = EIN, 3: BOASG
         $FLAG[334] = TRUE
      ;ENDFOLD
      ;FOLD Schritt 228 = T8 & A4039 ;%{SE}%MKUKATPVW %CVW_SPS %VST_CON %P 2:Schritt 228 = T8 & A4039, 3: ST_CON
         IF $TIMER_FLAG[8] AND $OUT[4039] THEN
            PREVSTEP = $APP_INT[5]
            $APP_INT[5] = 228
         ENDIF
      ;ENDFOLD
   ;ENDFOLD
   ;FOLD SCHRITT 228 -- STAT EZ1/SP1/KE1 Setzhub 2 -- ;%{P}%MKUKATPVW,%CSTEP,%VST_NR,%P 1:SCHRITT, 2:228, 3: STAT EZ1/SP1/KE1 Setzhub 2
      ;FOLD ;%{H}
         Case 228
      ;ENDFOLD
      ;FOLD -- Hilfsflag SK Programmwechsel -- ;%{SE}%MKUKATPVW %CVW_COM %VCOMMENT %P 2:-- Hilfsflag SK Programmwechsel --, 3: VW_COMMENT
      ;ENDFOLD
      ;FOLD F334 = AUS ;%{SE}%MKUKATPVW %CVW_SPS %VBOASG %P 2:F334 = AUS, 3: BOASG
         $FLAG[334] = FALSE
      ;ENDFOLD
      ;FOLD -- Zeit fuer Setzhub -- ;%{SE}%MKUKATPVW %CVW_COM %VCOMMENT %P 2:-- Zeit fuer Setzhub --, 3: VW_COMMENT
      ;ENDFOLD
      ;FOLD T8 ( EIN ) = -15[1/10Sek] ;%{SE}%MKUKATPVW %CVW_SPS %VTASG %P 2:T8 ( EIN ) = -15[1/10Sek], 3: TASG
         VW(#SET_TIME,TRUE,8,0,-15)
      ;ENDFOLD
      ;FOLD Schritt 229 = A4039 ;%{SE}%MKUKATPVW %CVW_SPS %VST_CON %P 2:Schritt 229 = A4039, 3: ST_CON
         IF $OUT[4039] THEN
            PREVSTEP = $APP_INT[5]
            $APP_INT[5] = 229
         ENDIF
      ;ENDFOLD
   ;ENDFOLD
   ;FOLD SCHRITT 229 -- STAT EZ3/SP3/KE3 Setzhub 2 -- ;%{P}%MKUKATPVW,%CSTEP,%VST_NR,%P 1:SCHRITT, 2:229, 3: STAT EZ3/SP3/KE3 Setzhub 2
      ;FOLD ;%{H}
         Case 229
      ;ENDFOLD
      ;FOLD -- Hilfsflag SK Programmwechsel -- ;%{SE}%MKUKATPVW %CVW_COM %VCOMMENT %P 2:-- Hilfsflag SK Programmwechsel --, 3: VW_COMMENT
      ;ENDFOLD
      ;FOLD F334 = AUS ;%{SE}%MKUKATPVW %CVW_SPS %VBOASG %P 2:F334 = AUS, 3: BOASG
         $FLAG[334] = FALSE
      ;ENDFOLD
      ;FOLD -- EZ3/SP3/KE3 schliessen -- ;%{SE}%MKUKATPVW %CVW_COM %VCOMMENT %P 2:-- EZ3/SP3/KE3 schliessen --, 3: VW_COMMENT
      ;ENDFOLD
      ;FOLD A1037 = AUS ;%{SE}%MKUKATPVW %CVW_SPS %VBOASG %P 2:A1037 = AUS, 3: BOASG
         $OUT[1037] = FALSE
      ;ENDFOLD
      ;FOLD -- EZ3/SP3 -- ;%{SE}%MKUKATPVW %CVW_COM %VCOMMENT %P 2:-- EZ3/SP3 --, 3: VW_COMMENT
      ;ENDFOLD
      ;FOLD A1038 = !F329 & !F122 & !F832 ;%{SE}%MKUKATPVW %CVW_SPS %VBOASG %P 2:A1038 = !F329 & !F122 & !F832, 3: BOASG
         $OUT[1038] = NOT $FLAG[329] AND NOT $FLAG[122] AND NOT $FLAG[832]
      ;ENDFOLD
      ;FOLD -- KE3 -- ;%{SE}%MKUKATPVW %CVW_COM %VCOMMENT %P 2:-- KE3 --, 3: VW_COMMENT
      ;ENDFOLD
      ;FOLD A1086 = !F329 & !F122 & F832 ;%{SE}%MKUKATPVW %CVW_SPS %VBOASG %P 2:A1086 = !F329 & !F122 & F832, 3: BOASG
         $OUT[1086] = NOT $FLAG[329] AND NOT $FLAG[122] AND $FLAG[832]
      ;ENDFOLD
      ;FOLD Schritt 230 = (!E1037 & E1038 & T8 + T9) & A4039 ;%{SE}%MKUKATPVW %CVW_SPS %VST_CON %P 2:Schritt 230 = (!E1037 & E1038 & T8 + T9) & A4039, 3: ST_CON
         IF (NOT $IN[1037] AND $IN[1038] AND $TIMER_FLAG[8] OR $TIMER_FLAG[9]) AND $OUT[4039] THEN
            PREVSTEP = $APP_INT[5]
            $APP_INT[5] = 230
         ENDIF
      ;ENDFOLD
   ;ENDFOLD
   ;FOLD SCHRITT 230 -- STAT EZ3/SP3/KE3 Setzhub 2 -- ;%{P}%MKUKATPVW,%CSTEP,%VST_NR,%P 1:SCHRITT, 2:230, 3: STAT EZ3/SP3/KE3 Setzhub 2
      ;FOLD ;%{H}
         Case 230
      ;ENDFOLD
      ;FOLD -- RSK Fehlerausgabe Kraftaufbau -- ;%{SE}%MKUKATPVW %CVW_COM %VCOMMENT %P 2:-- RSK Fehlerausgabe Kraftaufbau --, 3: VW_COMMENT
      ;ENDFOLD
      ;FOLD F325 = !E1038 & T9 ;%{SE}%MKUKATPVW %CVW_SPS %VBOASG %P 2:F325 = !E1038 & T9, 3: BOASG
         $FLAG[325] = NOT $IN[1038] AND $TIMER_FLAG[9]
      ;ENDFOLD
      ;FOLD F329 = T9 ;%{SE}%MKUKATPVW %CVW_SPS %VBOASG %P 2:F329 = T9, 3: BOASG
         $FLAG[329] = $TIMER_FLAG[9]
      ;ENDFOLD
      ;FOLD -- EZ3/SP3/KE3 SZ1 oeffnen -- ;%{SE}%MKUKATPVW %CVW_COM %VCOMMENT %P 2:-- EZ3/SP3/KE3 SZ1 oeffnen --, 3: VW_COMMENT
      ;ENDFOLD
      ;FOLD A1038 = AUS ;%{SE}%MKUKATPVW %CVW_SPS %VBOASG %P 2:A1038 = AUS, 3: BOASG
         $OUT[1038] = FALSE
      ;ENDFOLD
      ;FOLD A1086 = AUS ;%{SE}%MKUKATPVW %CVW_SPS %VBOASG %P 2:A1086 = AUS, 3: BOASG
         $OUT[1086] = FALSE
      ;ENDFOLD
      ;FOLD A1037 = EIN ;%{SE}%MKUKATPVW %CVW_SPS %VBOASG %P 2:A1037 = EIN, 3: BOASG
         $OUT[1037] = TRUE
      ;ENDFOLD
      ;FOLD -- Druckvorgabe SK3/EZ3/SP3/KE3 -- ;%{SE}%MKUKATPVW %CVW_COM %VCOMMENT %P 2:-- Druckvorgabe SK3/EZ3/SP3/KE3 --, 3: VW_COMMENT
      ;ENDFOLD
      ;FOLD F168 = F174 & !F832 ;%{SE}%MKUKATPVW %CVW_SPS %VBOASG %P 2:F168 = F174 & !F832, 3: BOASG
         $FLAG[168] = $FLAG[174] AND NOT $FLAG[832]
      ;ENDFOLD
      ;FOLD bin7 ( F168 ) = 41 ;%{SE}%MKUKATPVW %CVW_SPS %VARIASG %P 2:bin7 ( F168 ) = 41, 3: ARIASG
         VW(#BINOUT,$FLAG[168],7,41)
      ;ENDFOLD
      ;FOLD F168 = F175 & !F832 ;%{SE}%MKUKATPVW %CVW_SPS %VBOASG %P 2:F168 = F175 & !F832, 3: BOASG
         $FLAG[168] = $FLAG[175] AND NOT $FLAG[832]
      ;ENDFOLD
      ;FOLD bin7 ( F168 ) = 51 ;%{SE}%MKUKATPVW %CVW_SPS %VARIASG %P 2:bin7 ( F168 ) = 51, 3: ARIASG
         VW(#BINOUT,$FLAG[168],7,51)
      ;ENDFOLD
      ;FOLD F168 = AUS ;%{SE}%MKUKATPVW %CVW_SPS %VBOASG %P 2:F168 = AUS, 3: BOASG
         $FLAG[168] = FALSE
      ;ENDFOLD
      ;FOLD bin9 ( F174 ) = 41 ;%{SE}%MKUKATPVW %CVW_SPS %VARIASG %P 2:bin9 ( F174 ) = 41, 3: ARIASG
         VW(#BINOUT,$FLAG[174],9,41)
      ;ENDFOLD
      ;FOLD bin9 ( F175 ) = 51 ;%{SE}%MKUKATPVW %CVW_SPS %VARIASG %P 2:bin9 ( F175 ) = 51, 3: ARIASG
         VW(#BINOUT,$FLAG[175],9,51)
      ;ENDFOLD
      ;FOLD -- Wartezeit Programmwechsel SK -- ;%{SE}%MKUKATPVW %CVW_COM %VCOMMENT %P 2:-- Wartezeit Programmwechsel SK --, 3: VW_COMMENT
      ;ENDFOLD
      ;FOLD T8 ( !F334 ) = -2[1/10Sek] ;%{SE}%MKUKATPVW %CVW_SPS %VTASG %P 2:T8 ( !F334 ) = -2[1/10Sek], 3: TASG
         VW(#SET_TIME,NOT $FLAG[334],8,0,-2)
      ;ENDFOLD
      ;FOLD -- Hilfsflag SK Programmwechsel -- ;%{SE}%MKUKATPVW %CVW_COM %VCOMMENT %P 2:-- Hilfsflag SK Programmwechsel --, 3: VW_COMMENT
      ;ENDFOLD
      ;FOLD F334 = EIN ;%{SE}%MKUKATPVW %CVW_SPS %VBOASG %P 2:F334 = EIN, 3: BOASG
         $FLAG[334] = TRUE
      ;ENDFOLD
      ;FOLD Schritt 231 = T8 & A4039 ;%{SE}%MKUKATPVW %CVW_SPS %VST_CON %P 2:Schritt 231 = T8 & A4039, 3: ST_CON
         IF $TIMER_FLAG[8] AND $OUT[4039] THEN
            PREVSTEP = $APP_INT[5]
            $APP_INT[5] = 231
         ENDIF
      ;ENDFOLD
   ;ENDFOLD
   ;FOLD SCHRITT 231 -- STAT EZ3/SP3/KE3 Setzhub 2 -- ;%{P}%MKUKATPVW,%CSTEP,%VST_NR,%P 1:SCHRITT, 2:231, 3: STAT EZ3/SP3/KE3 Setzhub 2
      ;FOLD ;%{H}
         Case 231
      ;ENDFOLD
      ;FOLD -- Hilfsflag SK Programmwechsel -- ;%{SE}%MKUKATPVW %CVW_COM %VCOMMENT %P 2:-- Hilfsflag SK Programmwechsel --, 3: VW_COMMENT
      ;ENDFOLD
      ;FOLD F334 = AUS ;%{SE}%MKUKATPVW %CVW_SPS %VBOASG %P 2:F334 = AUS, 3: BOASG
         $FLAG[334] = FALSE
      ;ENDFOLD
      ;FOLD Schritt 116 = E1037 & !E1038 & A4039 ;%{SE}%MKUKATPVW %CVW_SPS %VST_CON %P 2:Schritt 116 = E1037 & !E1038 & A4039, 3: ST_CON
         IF $IN[1037] AND NOT $IN[1038] AND $OUT[4039] THEN
            PREVSTEP = $APP_INT[5]
            $APP_INT[5] = 116
         ENDIF
      ;ENDFOLD
   ;ENDFOLD
   ;FOLD SCHRITT 232 -- Reserviert -- ;%{P}%MKUKATPVW,%CSTEP,%VST_NR,%P 1:SCHRITT, 2:232, 3: Reserviert
      ;FOLD ;%{H}
         Case 232
      ;ENDFOLD
      ;FOLD 1:;%{SE} %MKUKATPVW
      ;ENDFOLD
   ;ENDFOLD
   ;FOLD SCHRITT 233 -- Reserviert -- ;%{P}%MKUKATPVW,%CSTEP,%VST_NR,%P 1:SCHRITT, 2:233, 3: Reserviert
      ;FOLD ;%{H}
         Case 233
      ;ENDFOLD
      ;FOLD 1:;%{SE} %MKUKATPVW
      ;ENDFOLD
   ;ENDFOLD
   ;FOLD SCHRITT 234 -- Reserviert -- ;%{P}%MKUKATPVW,%CSTEP,%VST_NR,%P 1:SCHRITT, 2:234, 3: Reserviert
      ;FOLD ;%{H}
         Case 234
      ;ENDFOLD
      ;FOLD 1:;%{SE} %MKUKATPVW
      ;ENDFOLD
   ;ENDFOLD
   ;FOLD SCHRITT 235 -- Reserviert -- ;%{P}%MKUKATPVW,%CSTEP,%VST_NR,%P 1:SCHRITT, 2:235, 3: Reserviert
      ;FOLD ;%{H}
         Case 235
      ;ENDFOLD
      ;FOLD 1:;%{SE} %MKUKATPVW
      ;ENDFOLD
   ;ENDFOLD
   ;FOLD SCHRITT 236 -- Reserviert -- ;%{P}%MKUKATPVW,%CSTEP,%VST_NR,%P 1:SCHRITT, 2:236, 3: Reserviert
      ;FOLD ;%{H}
         Case 236
      ;ENDFOLD
      ;FOLD 1:;%{SE} %MKUKATPVW
      ;ENDFOLD
   ;ENDFOLD
   ;FOLD SCHRITT 237 -- Reserviert -- ;%{P}%MKUKATPVW,%CSTEP,%VST_NR,%P 1:SCHRITT, 2:237, 3: Reserviert
      ;FOLD ;%{H}
         Case 237
      ;ENDFOLD
      ;FOLD 1:;%{SE} %MKUKATPVW
      ;ENDFOLD
   ;ENDFOLD
   ;FOLD SCHRITT 238 -- Reserviert -- ;%{P}%MKUKATPVW,%CSTEP,%VST_NR,%P 1:SCHRITT, 2:238, 3: Reserviert
      ;FOLD ;%{H}
         Case 238
      ;ENDFOLD
      ;FOLD 1:;%{SE} %MKUKATPVW
      ;ENDFOLD
   ;ENDFOLD
   ;FOLD SCHRITT 239 -- Reserviert -- ;%{P}%MKUKATPVW,%CSTEP,%VST_NR,%P 1:SCHRITT, 2:239, 3: Reserviert
      ;FOLD ;%{H}
         Case 239
      ;ENDFOLD
      ;FOLD 1:;%{SE} %MKUKATPVW
      ;ENDFOLD
   ;ENDFOLD
   ;FOLD SCHRITT 240 -- Reserviert -- ;%{P}%MKUKATPVW,%CSTEP,%VST_NR,%P 1:SCHRITT, 2:240, 3: Reserviert
      ;FOLD ;%{H}
         Case 240
      ;ENDFOLD
      ;FOLD 1:;%{SE} %MKUKATPVW
      ;ENDFOLD
   ;ENDFOLD
   ;FOLD SCHRITT 241 -- Reserviert -- ;%{P}%MKUKATPVW,%CSTEP,%VST_NR,%P 1:SCHRITT, 2:241, 3: Reserviert
      ;FOLD ;%{H}
         Case 241
      ;ENDFOLD
      ;FOLD 1:;%{SE} %MKUKATPVW
      ;ENDFOLD
   ;ENDFOLD
   ;FOLD SCHRITT 242 -- Reserviert -- ;%{P}%MKUKATPVW,%CSTEP,%VST_NR,%P 1:SCHRITT, 2:242, 3: Reserviert
      ;FOLD ;%{H}
         Case 242
      ;ENDFOLD
      ;FOLD 1:;%{SE} %MKUKATPVW
      ;ENDFOLD
   ;ENDFOLD
   ;FOLD SCHRITT 243 -- Reserviert -- ;%{P}%MKUKATPVW,%CSTEP,%VST_NR,%P 1:SCHRITT, 2:243, 3: Reserviert
      ;FOLD ;%{H}
         Case 243
      ;ENDFOLD
      ;FOLD 1:;%{SE} %MKUKATPVW
      ;ENDFOLD
   ;ENDFOLD
   ;FOLD SCHRITT 244 -- Reserviert -- ;%{P}%MKUKATPVW,%CSTEP,%VST_NR,%P 1:SCHRITT, 2:244, 3: Reserviert
      ;FOLD ;%{H}
         Case 244
      ;ENDFOLD
      ;FOLD 1:;%{SE} %MKUKATPVW
      ;ENDFOLD
   ;ENDFOLD
   ;FOLD SCHRITT 245 -- Reserviert -- ;%{P}%MKUKATPVW,%CSTEP,%VST_NR,%P 1:SCHRITT, 2:245, 3: Reserviert
      ;FOLD ;%{H}
         Case 245
      ;ENDFOLD
      ;FOLD 1:;%{SE} %MKUKATPVW
      ;ENDFOLD
   ;ENDFOLD
   ;FOLD SCHRITT 246 -- Reserviert -- ;%{P}%MKUKATPVW,%CSTEP,%VST_NR,%P 1:SCHRITT, 2:246, 3: Reserviert
      ;FOLD ;%{H}
         Case 246
      ;ENDFOLD
      ;FOLD 1:;%{SE} %MKUKATPVW
      ;ENDFOLD
   ;ENDFOLD
   ;FOLD SCHRITT 247 -- Reserviert -- ;%{P}%MKUKATPVW,%CSTEP,%VST_NR,%P 1:SCHRITT, 2:247, 3: Reserviert
      ;FOLD ;%{H}
         Case 247
      ;ENDFOLD
      ;FOLD 1:;%{SE} %MKUKATPVW
      ;ENDFOLD
   ;ENDFOLD
   ;FOLD SCHRITT 248 -- Reserviert -- ;%{P}%MKUKATPVW,%CSTEP,%VST_NR,%P 1:SCHRITT, 2:248, 3: Reserviert
      ;FOLD ;%{H}
         Case 248
      ;ENDFOLD
      ;FOLD 1:;%{SE} %MKUKATPVW
      ;ENDFOLD
   ;ENDFOLD
   ;FOLD SCHRITT 249 -- Reserviert -- ;%{P}%MKUKATPVW,%CSTEP,%VST_NR,%P 1:SCHRITT, 2:249, 3: Reserviert
      ;FOLD ;%{H}
         Case 249
      ;ENDFOLD
      ;FOLD 1:;%{SE} %MKUKATPVW
      ;ENDFOLD
   ;ENDFOLD
   ;FOLD SCHRITT 250 -- MB1 Fraesen mit KFB1 # Start -- ;%{P}%MKUKATPVW,%CSTEP,%VST_NR,%P 1:SCHRITT, 2:250, 3: MB1 Fraesen mit KFB1 # Start
      ;FOLD ;%{H}
         Case 250
      ;ENDFOLD
      ;FOLD -- RSK gestartet -- ;%{SE}%MKUKATPVW %CVW_COM %VCOMMENT %P 2:-- RSK gestartet --, 3: VW_COMMENT
      ;ENDFOLD
      ;FOLD F321 = AUS ;%{SE}%MKUKATPVW %CVW_SPS %VBOASG %P 2:F321 = AUS, 3: BOASG
         $FLAG[321] = FALSE
      ;ENDFOLD
      ;FOLD F322 = AUS ;%{SE}%MKUKATPVW %CVW_SPS %VBOASG %P 2:F322 = AUS, 3: BOASG
         $FLAG[322] = FALSE
      ;ENDFOLD
      ;FOLD F323 = AUS ;%{SE}%MKUKATPVW %CVW_SPS %VBOASG %P 2:F323 = AUS, 3: BOASG
         $FLAG[323] = FALSE
      ;ENDFOLD
      ;FOLD F324 = AUS ;%{SE}%MKUKATPVW %CVW_SPS %VBOASG %P 2:F324 = AUS, 3: BOASG
         $FLAG[324] = FALSE
      ;ENDFOLD
      ;FOLD F325 = AUS ;%{SE}%MKUKATPVW %CVW_SPS %VBOASG %P 2:F325 = AUS, 3: BOASG
         $FLAG[325] = FALSE
      ;ENDFOLD
      ;FOLD F326 = AUS ;%{SE}%MKUKATPVW %CVW_SPS %VBOASG %P 2:F326 = AUS, 3: BOASG
         $FLAG[326] = FALSE
      ;ENDFOLD
      ;FOLD F327 = AUS ;%{SE}%MKUKATPVW %CVW_SPS %VBOASG %P 2:F327 = AUS, 3: BOASG
         $FLAG[327] = FALSE
      ;ENDFOLD
      ;FOLD F329 = AUS ;%{SE}%MKUKATPVW %CVW_SPS %VBOASG %P 2:F329 = AUS, 3: BOASG
         $FLAG[329] = FALSE
      ;ENDFOLD
      ;FOLD -- MB1 Zaehler -- ;%{SE}%MKUKATPVW %CVW_COM %VCOMMENT %P 2:-- MB1 Zaehler --, 3: VW_COMMENT
      ;ENDFOLD
      ;FOLD F186 = AUS ;%{SE}%MKUKATPVW %CVW_SPS %VBOASG %P 2:F186 = AUS, 3: BOASG
         $FLAG[186] = FALSE
      ;ENDFOLD
      ;FOLD F187 = AUS ;%{SE}%MKUKATPVW %CVW_SPS %VBOASG %P 2:F187 = AUS, 3: BOASG
         $FLAG[187] = FALSE
      ;ENDFOLD
      ;FOLD F188 = AUS ;%{SE}%MKUKATPVW %CVW_SPS %VBOASG %P 2:F188 = AUS, 3: BOASG
         $FLAG[188] = FALSE
      ;ENDFOLD
      ;FOLD F189 = AUS ;%{SE}%MKUKATPVW %CVW_SPS %VBOASG %P 2:F189 = AUS, 3: BOASG
         $FLAG[189] = FALSE
      ;ENDFOLD
      ;FOLD F190 = AUS ;%{SE}%MKUKATPVW %CVW_SPS %VBOASG %P 2:F190 = AUS, 3: BOASG
         $FLAG[190] = FALSE
      ;ENDFOLD
      ;FOLD F191 = AUS ;%{SE}%MKUKATPVW %CVW_SPS %VBOASG %P 2:F191 = AUS, 3: BOASG
         $FLAG[191] = FALSE
      ;ENDFOLD
      ;FOLD -- Hilfsflags Funktionstest KF Motor -- ;%{SE}%MKUKATPVW %CVW_COM %VCOMMENT %P 2:-- Hilfsflags Funktionstest KF Motor --, 3: VW_COMMENT
      ;ENDFOLD
      ;FOLD F312 = AUS ;%{SE}%MKUKATPVW %CVW_SPS %VBOASG %P 2:F312 = AUS, 3: BOASG
         $FLAG[312] = FALSE
      ;ENDFOLD
      ;FOLD F313 = AUS ;%{SE}%MKUKATPVW %CVW_SPS %VBOASG %P 2:F313 = AUS, 3: BOASG
         $FLAG[313] = FALSE
      ;ENDFOLD
      ;FOLD -- Serviceprogramm Fraesen an MB1 -- ;%{SE}%MKUKATPVW %CVW_COM %VCOMMENT %P 2:-- Serviceprogramm Fraesen an MB1 --, 3: VW_COMMENT
      ;ENDFOLD
      ;FOLD bin7 ( EIN ) = 23 ;%{SE}%MKUKATPVW %CVW_SPS %VARIASG %P 2:bin7 ( EIN ) = 23, 3: ARIASG
         VW(#BINOUT,TRUE,7,23)
      ;ENDFOLD
      ;FOLD -- Wartezeit Programmwechsel SK -- ;%{SE}%MKUKATPVW %CVW_COM %VCOMMENT %P 2:-- Wartezeit Programmwechsel SK --, 3: VW_COMMENT
      ;ENDFOLD
      ;FOLD T8 ( !F334 ) = -2[1/10Sek] ;%{SE}%MKUKATPVW %CVW_SPS %VTASG %P 2:T8 ( !F334 ) = -2[1/10Sek], 3: TASG
         VW(#SET_TIME,NOT $FLAG[334],8,0,-2)
      ;ENDFOLD
      ;FOLD -- Hilfsflag SK Programmwechsel -- ;%{SE}%MKUKATPVW %CVW_COM %VCOMMENT %P 2:-- Hilfsflag SK Programmwechsel --, 3: VW_COMMENT
      ;ENDFOLD
      ;FOLD F334 = EIN ;%{SE}%MKUKATPVW %CVW_SPS %VBOASG %P 2:F334 = EIN, 3: BOASG
         $FLAG[334] = TRUE
      ;ENDFOLD
      ;FOLD -- Stat. MB 1 beim Fraesen -- ;%{SE}%MKUKATPVW %CVW_COM %VCOMMENT %P 2:-- Stat. MB 1 beim Fraesen --, 3: VW_COMMENT
      ;ENDFOLD
      ;FOLD A1812 = EIN ;%{SE}%MKUKATPVW %CVW_SPS %VBOASG %P 2:A1812 = EIN, 3: BOASG
         $OUT[1812] = TRUE
      ;ENDFOLD
      ;FOLD Schritt 251 = T8 & A4039 ;%{SE}%MKUKATPVW %CVW_SPS %VST_CON %P 2:Schritt 251 = T8 & A4039, 3: ST_CON
         IF $TIMER_FLAG[8] AND $OUT[4039] THEN
            PREVSTEP = $APP_INT[5]
            $APP_INT[5] = 251
         ENDIF
      ;ENDFOLD
   ;ENDFOLD
   ;FOLD SCHRITT 251 -- MB1 Fraesen mit KFB1 -- ;%{P}%MKUKATPVW,%CSTEP,%VST_NR,%P 1:SCHRITT, 2:251, 3: MB1 Fraesen mit KFB1
      ;FOLD ;%{H}
         Case 251
      ;ENDFOLD
      ;FOLD -- Ueberwachungszeit KFB1 EIN -- ;%{SE}%MKUKATPVW %CVW_COM %VCOMMENT %P 2:-- Ueberwachungszeit KFB1 EIN --, 3: VW_COMMENT
      ;ENDFOLD
      ;FOLD -- Hilfsflag SK Programmwechsel -- ;%{SE}%MKUKATPVW %CVW_COM %VCOMMENT %P 2:-- Hilfsflag SK Programmwechsel --, 3: VW_COMMENT
      ;ENDFOLD
      ;FOLD F334 = AUS ;%{SE}%MKUKATPVW %CVW_SPS %VBOASG %P 2:F334 = AUS, 3: BOASG
         $FLAG[334] = FALSE
      ;ENDFOLD
      ;FOLD T7 ( EIN ) = -30[1/10Sek] ;%{SE}%MKUKATPVW %CVW_SPS %VTASG %P 2:T7 ( EIN ) = -30[1/10Sek], 3: TASG
         VW(#SET_TIME,TRUE,7,0,-30)
      ;ENDFOLD
      ;FOLD -- KFB1 einschalten -- ;%{SE}%MKUKATPVW %CVW_COM %VCOMMENT %P 2:-- KFB1 einschalten --, 3: VW_COMMENT
      ;ENDFOLD
      ;FOLD i1 (EIN) = 0 ;%{SE}%MKUKATPVW %CVW_SPS %VARIASG %P 2:i1 (EIN) = 0, 3: ARIASG
         VW(#COUNTER,TRUE,1,0)
      ;ENDFOLD
      ;FOLD A1154 = EIN ;%{SE}%MKUKATPVW %CVW_SPS %VBOASG %P 2:A1154 = EIN, 3: BOASG
         $OUT[1154] = TRUE
      ;ENDFOLD
      ;FOLD Schritt 252 = A4039 ;%{SE}%MKUKATPVW %CVW_SPS %VST_CON %P 2:Schritt 252 = A4039, 3: ST_CON
         IF $OUT[4039] THEN
            PREVSTEP = $APP_INT[5]
            $APP_INT[5] = 252
         ENDIF
      ;ENDFOLD
   ;ENDFOLD
   ;FOLD SCHRITT 252 -- MB1 Fraesen mit KFB1 -- ;%{P}%MKUKATPVW,%CSTEP,%VST_NR,%P 1:SCHRITT, 2:252, 3: MB1 Fraesen mit KFB1
      ;FOLD ;%{H}
         Case 252
      ;ENDFOLD
      ;FOLD -- Funktionstest KF Motor -- ;%{SE}%MKUKATPVW %CVW_COM %VCOMMENT %P 2:-- Funktionstest KF Motor --, 3: VW_COMMENT
      ;ENDFOLD
      ;FOLD F312 = EIN ;%{SE}%MKUKATPVW %CVW_SPS %VBOASG %P 2:F312 = EIN, 3: BOASG
         $FLAG[312] = TRUE
      ;ENDFOLD
      ;FOLD F313 = i1 > 2 ;%{SE}%MKUKATPVW %CVW_SPS %VBOCMP %P 2:F313 = i1 > 2, 3: BOCMP
         $FLAG[313] = $COUNT_I[1] > 2
      ;ENDFOLD
      ;FOLD Schritt 253 = (F313 + T7) & A4039 ;%{SE}%MKUKATPVW %CVW_SPS %VST_CON %P 2:Schritt 253 = (F313 + T7) & A4039, 3: ST_CON
         IF ($FLAG[313] OR $TIMER_FLAG[7]) AND $OUT[4039] THEN
            PREVSTEP = $APP_INT[5]
            $APP_INT[5] = 253
         ENDIF
      ;ENDFOLD
   ;ENDFOLD
   ;FOLD SCHRITT 253 -- MB1 Fraesen mit KFB1 -- ;%{P}%MKUKATPVW,%CSTEP,%VST_NR,%P 1:SCHRITT, 2:253, 3: MB1 Fraesen mit KFB1
      ;FOLD ;%{H}
         Case 253
      ;ENDFOLD
      ;FOLD F312 = AUS ;%{SE}%MKUKATPVW %CVW_SPS %VBOASG %P 2:F312 = AUS, 3: BOASG
         $FLAG[312] = FALSE
      ;ENDFOLD
      ;FOLD -- Ueberwachungszeit KSB1 schwenken -- ;%{SE}%MKUKATPVW %CVW_COM %VCOMMENT %P 2:-- Ueberwachungszeit KSB1 schwenken --, 3: VW_COMMENT
      ;ENDFOLD
      ;FOLD t8 ( EIN ) = -100[1/10Sek] ;%{SE}%MKUKATPVW %CVW_SPS %VTASG %P 2:t8 ( EIN ) = -100[1/10Sek], 3: TASG
         VW(#SET_TIME,TRUE,8,0,-100)
      ;ENDFOLD
      ;FOLD Schritt 254 = A4039 ;%{SE}%MKUKATPVW %CVW_SPS %VST_CON %P 2:Schritt 254 = A4039, 3: ST_CON
         IF $OUT[4039] THEN
            PREVSTEP = $APP_INT[5]
            $APP_INT[5] = 254
         ENDIF
      ;ENDFOLD
   ;ENDFOLD
   ;FOLD SCHRITT 254 -- MB1 Fraesen mit KFB1-- ;%{P}%MKUKATPVW,%CSTEP,%VST_NR,%P 1:SCHRITT, 2:254, 3: MB1 Fraesen mit KFB1
      ;FOLD ;%{H}
         Case 254
      ;ENDFOLD
      ;FOLD -- RSK Fehlerausgabe KFB1 Initiator/Motor -- ;%{SE}%MKUKATPVW %CVW_COM %VCOMMENT %P 2:-- RSK Fehlerausgabe KFB1 Initiator/Motor --, 3: VW_COMMENT
      ;ENDFOLD
      ;FOLD F322 = !F313 ;%{SE}%MKUKATPVW %CVW_SPS %VBOASG %P 2:F322 = !F313, 3: BOASG
         $FLAG[322] = NOT $FLAG[313]
      ;ENDFOLD
      ;FOLD -- RSK Fehlerausgabe KSB1 Ruhest. -- ;%{SE}%MKUKATPVW %CVW_COM %VCOMMENT %P 2:-- RSK Fehlerausgabe KSB1 Ruhest. --, 3: VW_COMMENT
      ;ENDFOLD
      ;FOLD F323 = !E1156 & F324 + !E1156 & F328 ;%{SE}%MKUKATPVW %CVW_SPS %VBOASG %P 2:F323 = !E1156 & F324 + !E1156 & F328, 3: BOASG
         $FLAG[323] = NOT $IN[1156] AND $FLAG[324] OR NOT $IN[1156] AND $FLAG[328]
      ;ENDFOLD
      ;FOLD -- RSK Sammelstoerung -- ;%{SE}%MKUKATPVW %CVW_COM %VCOMMENT %P 2:-- RSK Sammelstoerung --, 3: VW_COMMENT
      ;ENDFOLD
      ;FOLD F329 = F322 + F323 ;%{SE}%MKUKATPVW %CVW_SPS %VBOASG %P 2:F329 = F322 + F323, 3: BOASG
         $FLAG[329] = $FLAG[322] OR $FLAG[323]
      ;ENDFOLD
      ;FOLD t7 ( EIN ) = STOP ;%{SE}%MKUKATPVW %CVW_SPS %VTSTOP %P 2:t7 ( EIN ) = STOP, 3: TSTOP
         VW(#SET_TIME,TRUE,7,1,0)
      ;ENDFOLD
      ;FOLD A1154 = !F322 & !F323 ;%{SE}%MKUKATPVW %CVW_SPS %VBOASG %P 2:A1154 = !F322 & !F323, 3: BOASG
         $OUT[1154] = NOT $FLAG[322] AND NOT $FLAG[323]
      ;ENDFOLD
      ;FOLD -- KFB1 Versetzeinheit vor -- ;%{SE}%MKUKATPVW %CVW_COM %VCOMMENT %P 2:-- KFB1 Versetzeinheit vor --, 3: VW_COMMENT
      ;ENDFOLD
      ;FOLD A1155 = !F322 & !F323 & F564 ;%{SE}%MKUKATPVW %CVW_SPS %VBOASG %P 2:A1155 = !F322 & !F323 & F564, 3: BOASG
         $OUT[1155] = NOT $FLAG[322] AND NOT $FLAG[323] AND $FLAG[564]
      ;ENDFOLD
      ;FOLD Schritt 255 = (!F322 & !F323 & (E1155 & F564 + !E1155 & !F564) + T8) & A4039 ;%{SE}%MKUKATPVW %CVW_SPS %VST_CON %P 2:Schritt 255 = (!F322 & !F323 & (E1155 & F564 + !E1155 & !F564) + T8) & A4039, 3: ST_CON
         IF (NOT $FLAG[322] AND NOT $FLAG[323] AND ($IN[1155] AND $FLAG[564] OR NOT $IN[1155] AND NOT $FLAG[564]) OR $TIMER_FLAG[8]) AND $OUT[4039] THEN
            PREVSTEP = $APP_INT[5]
            $APP_INT[5] = 255
         ENDIF
      ;ENDFOLD
      ;FOLD Schritt 271 = (F322 + F323) & !F324 & !F328 & A4039 ;%{SE}%MKUKATPVW %CVW_SPS %VST_CON %P 2:Schritt 271 = (F322 + F323) & !F324 & !F328 & A4039, 3: ST_CON
         IF ($FLAG[322] OR $FLAG[323]) AND NOT $FLAG[324] AND NOT $FLAG[328] AND $OUT[4039] THEN
            PREVSTEP = $APP_INT[5]
            $APP_INT[5] = 271
         ENDIF
      ;ENDFOLD
   ;ENDFOLD
   ;FOLD SCHRITT 255 -- MB1 Fraesen mit KFB1 -- ;%{P}%MKUKATPVW,%CSTEP,%VST_NR,%P 1:SCHRITT, 2:255, 3: MB1 Fraesen mit KFB1
      ;FOLD ;%{H}
         Case 255
      ;ENDFOLD
      ;FOLD F329 = T8 ;%{SE}%MKUKATPVW %CVW_SPS %VBOASG %P 2:F329 = T8, 3: BOASG
         $FLAG[329] = $TIMER_FLAG[8]
      ;ENDFOLD
      ;FOLD F324 = AUS ;%{SE}%MKUKATPVW %CVW_SPS %VBOASG %P 2:F324 = AUS, 3: BOASG
         $FLAG[324] = FALSE
      ;ENDFOLD
      ;FOLD F328 = AUS ;%{SE}%MKUKATPVW %CVW_SPS %VBOASG %P 2:F328 = AUS, 3: BOASG
         $FLAG[328] = FALSE
      ;ENDFOLD
      ;FOLD -- KSB1 in Arbeitsstellung schwenken -- ;%{SE}%MKUKATPVW %CVW_COM %VCOMMENT %P 2:-- KSB1 in Arbeitsstellung schwenken --, 3: VW_COMMENT
      ;ENDFOLD
      ;FOLD A1163 = E1798 & (E1155 & F564 + !E1155 & !F564) ;%{SE}%MKUKATPVW %CVW_SPS %VBOASG %P 2:A1163 = E1798 & (E1155 & F564 + !E1155 & !F564), 3: BOASG
         $OUT[1163] = $IN[1798] AND ($IN[1155] AND $FLAG[564] OR NOT $IN[1155] AND NOT $FLAG[564])
      ;ENDFOLD
      ;FOLD Schritt 253 = !E1155 & F564 & T8 & (E26 + E27) & A4039 ;%{SE}%MKUKATPVW %CVW_SPS %VST_CON %P 2:Schritt 253 = !E1155 & F564 & T8 & (E26 + E27) & A4039, 3: ST_CON
         IF NOT $IN[1155] AND $FLAG[564] AND $TIMER_FLAG[8] AND ($IN[26] OR $IN[27]) AND $OUT[4039] THEN
            PREVSTEP = $APP_INT[5]
            $APP_INT[5] = 253
         ENDIF
      ;ENDFOLD
      ;FOLD Schritt 256 = E1798 & (A1163 + E1157) & A4039 ;%{SE}%MKUKATPVW %CVW_SPS %VST_CON %P 2:Schritt 256 = E1798 & (A1163 + E1157) & A4039, 3: ST_CON
         IF $IN[1798] AND ($OUT[1163] OR $IN[1157]) AND $OUT[4039] THEN
            PREVSTEP = $APP_INT[5]
            $APP_INT[5] = 256
         ENDIF
      ;ENDFOLD
   ;ENDFOLD
   ;FOLD SCHRITT 256 -- MB1 Fraesen mit KFB1-- ;%{P}%MKUKATPVW,%CSTEP,%VST_NR,%P 1:SCHRITT, 2:256, 3: MB1 Fraesen mit KFB1
      ;FOLD ;%{H}
         Case 256
      ;ENDFOLD
      ;FOLD -- RSK Fehlerausgabe KF Versetzeinheit -- ;%{SE}%MKUKATPVW %CVW_COM %VCOMMENT %P 2:-- RSK Fehlerausgabe KF Versetzeinheit --, 3: VW_COMMENT
      ;ENDFOLD
      ;FOLD F328 = !E1155 & F564 & !F324 ;%{SE}%MKUKATPVW %CVW_SPS %VBOASG %P 2:F328 = !E1155 & F564 & !F324, 3: BOASG
         $FLAG[328] = NOT $IN[1155] AND $FLAG[564] AND NOT $FLAG[324]
      ;ENDFOLD
      ;FOLD -- RSK Fehlerausgabe KSB1 Arbeitsstellung -- ;%{SE}%MKUKATPVW %CVW_COM %VCOMMENT %P 2:-- RSK Fehlerausgabe KSB1 Arbeitsstellung --, 3: VW_COMMENT
      ;ENDFOLD
      ;FOLD F324 = (!E1157 + E1159) & T8 & (E1155 + !F564) + F324 ;%{SE}%MKUKATPVW %CVW_SPS %VBOASG %P 2:F324 = (!E1157 + E1159) & T8 & (E1155 + !F564) + F324, 3: BOASG
         $FLAG[324] = (NOT $IN[1157] OR $IN[1159]) AND $TIMER_FLAG[8] AND ($IN[1155] OR NOT $FLAG[564]) OR $FLAG[324]
      ;ENDFOLD
      ;FOLD -- RSK Sammelstoerung -- ;%{SE}%MKUKATPVW %CVW_COM %VCOMMENT %P 2:-- RSK Sammelstoerung --, 3: VW_COMMENT
      ;ENDFOLD
      ;FOLD F329 = F324 + F328 ;%{SE}%MKUKATPVW %CVW_SPS %VBOASG %P 2:F329 = F324 + F328, 3: BOASG
         $FLAG[329] = $FLAG[324] OR $FLAG[328]
      ;ENDFOLD
      ;FOLD A1154 = !F324 & !F328 ;%{SE}%MKUKATPVW %CVW_SPS %VBOASG %P 2:A1154 = !F324 & !F328, 3: BOASG
         $OUT[1154] = NOT $FLAG[324] AND NOT $FLAG[328]
      ;ENDFOLD
      ;FOLD A1155 = !F324 & !F328 & F564 ;%{SE}%MKUKATPVW %CVW_SPS %VBOASG %P 2:A1155 = !F324 & !F328 & F564, 3: BOASG
         $OUT[1155] = NOT $FLAG[324] AND NOT $FLAG[328] AND $FLAG[564]
      ;ENDFOLD
      ;FOLD -- Ueberwachungszeit EZ3/SP3/KE3 schliessen -- ;%{SE}%MKUKATPVW %CVW_COM %VCOMMENT %P 2:-- Ueberwachungszeit EZ3/SP3/KE3 schliessen --, 3: VW_COMMENT
      ;ENDFOLD
      ;FOLD t9 ( EIN ) = -120[1/10Sek] ;%{SE}%MKUKATPVW %CVW_SPS %VTASG %P 2:t9 ( EIN ) = -120[1/10Sek], 3: TASG
         VW(#SET_TIME,TRUE,9,0,-120)
      ;ENDFOLD
      ;FOLD -- Verweilzeit Versetzeinheit Rueck -- ;%{SE}%MKUKATPVW %CVW_COM %VCOMMENT %P 2:-- Verweilzeit Versetzeinheit Rueck --, 3: VW_COMMENT
      ;ENDFOLD
      ;FOLD t11 ( EIN ) = i24[1/10Sek] ;%{SE}%MKUKATPVW %CVW_SPS %VTASG %P 2:t11 ( EIN ) = i24[1/10Sek], 3: TASG
         VW(#SET_TIME,TRUE,11,0,$COUNT_I[24])
      ;ENDFOLD
      ;FOLD Schritt 251 = (F324 + F328) & (E26 + E27) & A4039 ;%{SE}%MKUKATPVW %CVW_SPS %VST_CON %P 2:Schritt 251 = (F324 + F328) & (E26 + E27) & A4039, 3: ST_CON
         IF ($FLAG[324] OR $FLAG[328]) AND ($IN[26] OR $IN[27]) AND $OUT[4039] THEN
            PREVSTEP = $APP_INT[5]
            $APP_INT[5] = 251
         ENDIF
      ;ENDFOLD
      ;FOLD Schritt 257 = !F324 & !F328 & E1157 & A4039 ;%{SE}%MKUKATPVW %CVW_SPS %VST_CON %P 2:Schritt 257 = !F324 & !F328 & E1157 & A4039, 3: ST_CON
         IF NOT $FLAG[324] AND NOT $FLAG[328] AND $IN[1157] AND $OUT[4039] THEN
            PREVSTEP = $APP_INT[5]
            $APP_INT[5] = 257
         ENDIF
      ;ENDFOLD
   ;ENDFOLD
   ;FOLD SCHRITT 257 -- MB1 Fraesen mit KFB1 -- ;%{P}%MKUKATPVW,%CSTEP,%VST_NR,%P 1:SCHRITT, 2:257, 3: MB1 Fraesen mit KFB1
      ;FOLD ;%{H}
         Case 257
      ;ENDFOLD
      ;FOLD -- Umdreh. KF setzen -- ;%{SE}%MKUKATPVW %CVW_COM %VCOMMENT %P 2:-- Umdreh. KF setzen --, 3: VW_COMMENT
      ;ENDFOLD
      ;FOLD i1 ( EIN ) = 0 ;%{SE}%MKUKATPVW %CVW_SPS %VARIASG %P 2:i1 ( EIN ) = 0, 3: ARIASG
         VW(#COUNTER,TRUE,1,0)
      ;ENDFOLD
      ;FOLD F190 = AUS ;%{SE}%MKUKATPVW %CVW_SPS %VBOASG %P 2:F190 = AUS, 3: BOASG
         $FLAG[190] = FALSE
      ;ENDFOLD
      ;FOLD F312 = AUS ;%{SE}%MKUKATPVW %CVW_SPS %VBOASG %P 2:F312 = AUS, 3: BOASG
         $FLAG[312] = FALSE
      ;ENDFOLD
      ;FOLD F313 = AUS ;%{SE}%MKUKATPVW %CVW_SPS %VBOASG %P 2:F313 = AUS, 3: BOASG
         $FLAG[313] = FALSE
      ;ENDFOLD
      ;FOLD F324 = AUS ;%{SE}%MKUKATPVW %CVW_SPS %VBOASG %P 2:F324 = AUS, 3: BOASG
         $FLAG[324] = FALSE
      ;ENDFOLD
      ;FOLD F328 = AUS ;%{SE}%MKUKATPVW %CVW_SPS %VBOASG %P 2:F328 = AUS, 3: BOASG
         $FLAG[328] = FALSE
      ;ENDFOLD
      ;FOLD -- KSB1 in Arbeitsstellung schwenken AUS -- ;%{SE}%MKUKATPVW %CVW_COM %VCOMMENT %P 2:-- KSB1 in Arbeitsstellung schwenken AUS --, 3: VW_COMMENT
      ;ENDFOLD
      ;FOLD A1163 = AUS ;%{SE}%MKUKATPVW %CVW_SPS %VBOASG %P 2:A1163 = AUS, 3: BOASG
         $OUT[1163] = FALSE
      ;ENDFOLD
      ;FOLD -- KFB1 einschalten nach Fehler -- ;%{SE}%MKUKATPVW %CVW_COM %VCOMMENT %P 2:-- KFB1 einschalten nach Fehler --, 3: VW_COMMENT
      ;ENDFOLD
      ;FOLD A1154 = EIN ;%{SE}%MKUKATPVW %CVW_SPS %VBOASG %P 2:A1154 = EIN, 3: BOASG
         $OUT[1154] = TRUE
      ;ENDFOLD
      ;FOLD -- KFB1 Versetzeinheit rueck -- ;%{SE}%MKUKATPVW %CVW_COM %VCOMMENT %P 2:-- KFB1 Versetzeinheit rueck --, 3: VW_COMMENT
      ;ENDFOLD
      ;FOLD A1155 = AUS ;%{SE}%MKUKATPVW %CVW_SPS %VBOASG %P 2:A1155 = AUS, 3: BOASG
         $OUT[1155] = FALSE
      ;ENDFOLD
      ;FOLD Schritt 258 = T11 & A4039 ;%{SE}%MKUKATPVW %CVW_SPS %VST_CON %P 2:Schritt 258 = T11 & A4039, 3: ST_CON
         IF $TIMER_FLAG[11] AND $OUT[4039] THEN
            PREVSTEP = $APP_INT[5]
            $APP_INT[5] = 258
         ENDIF
      ;ENDFOLD
   ;ENDFOLD
   ;FOLD SCHRITT 258 -- MB1 Fraesen mit KFB1-- ;%{P}%MKUKATPVW,%CSTEP,%VST_NR,%P 1:SCHRITT, 2:258, 3: MB1 Fraesen mit KFB1
      ;FOLD ;%{H}
         Case 258
      ;ENDFOLD
      ;FOLD t11 ( EIN ) = STOP ;%{SE}%MKUKATPVW %CVW_SPS %VTSTOP %P 2:t11 ( EIN ) = STOP, 3: TSTOP
         VW(#SET_TIME,TRUE,11,1,0)
      ;ENDFOLD
      ;FOLD -- MB1 schliessen -- ;%{SE}%MKUKATPVW %CVW_COM %VCOMMENT %P 2:-- MB1 schliessen --, 3: VW_COMMENT
      ;ENDFOLD
      ;FOLD A1798 = AUS ;%{SE}%MKUKATPVW %CVW_SPS %VBOASG %P 2:A1798 = AUS, 3: BOASG
         $OUT[1798] = FALSE
      ;ENDFOLD
      ;FOLD A1802 = EIN ;%{SE}%MKUKATPVW %CVW_SPS %VBOASG %P 2:A1802 = EIN, 3: BOASG
         $OUT[1802] = TRUE
      ;ENDFOLD
      ;FOLD -- AUSBLASEN  EIN -- ;%{SE}%MKUKATPVW %CVW_COM %VCOMMENT %P 2:-- AUSBLASEN  EIN --, 3: VW_COMMENT
      ;ENDFOLD
      ;FOLD A1166 = EIN ;%{SE}%MKUKATPVW %CVW_SPS %VBOASG %P 2:A1166 = EIN, 3: BOASG
         $OUT[1166] = TRUE
      ;ENDFOLD
      ;FOLD Schritt 259 = (!E1798 & E1802 + T9) & A4039 ;%{SE}%MKUKATPVW %CVW_SPS %VST_CON %P 2:Schritt 259 = (!E1798 & E1802 + T9) & A4039, 3: ST_CON
         IF (NOT $IN[1798] AND $IN[1802] OR $TIMER_FLAG[9]) AND $OUT[4039] THEN
            PREVSTEP = $APP_INT[5]
            $APP_INT[5] = 259
         ENDIF
      ;ENDFOLD
   ;ENDFOLD
   ;FOLD SCHRITT 259 -- MB1 Fraesen mit KFB1-- ;%{P}%MKUKATPVW,%CSTEP,%VST_NR,%P 1:SCHRITT, 2:259, 3: MB1 Fraesen mit KFB1
      ;FOLD ;%{H}
         Case 259
      ;ENDFOLD
      ;FOLD -- RSK Fehlerausgabe Kraftaufbau -- ;%{SE}%MKUKATPVW %CVW_COM %VCOMMENT %P 2:-- RSK Fehlerausgabe Kraftaufbau --, 3: VW_COMMENT
      ;ENDFOLD
      ;FOLD F325 = T9 ;%{SE}%MKUKATPVW %CVW_SPS %VBOASG %P 2:F325 = T9, 3: BOASG
         $FLAG[325] = $TIMER_FLAG[9]
      ;ENDFOLD
      ;FOLD -- RSK Sammelstoerung -- ;%{SE}%MKUKATPVW %CVW_COM %VCOMMENT %P 2:-- RSK Sammelstoerung --, 3: VW_COMMENT
      ;ENDFOLD
      ;FOLD F329 = F325 ;%{SE}%MKUKATPVW %CVW_SPS %VBOASG %P 2:F329 = F325, 3: BOASG
         $FLAG[329] = $FLAG[325]
      ;ENDFOLD
      ;FOLD -- KFB1 abschalten bei Fehler -- ;%{SE}%MKUKATPVW %CVW_COM %VCOMMENT %P 2:-- KFB1 abschalten bei Fehler --, 3: VW_COMMENT
      ;ENDFOLD
      ;FOLD A1154 = !T9 ;%{SE}%MKUKATPVW %CVW_SPS %VBOASG %P 2:A1154 = !T9, 3: BOASG
         $OUT[1154] = NOT $TIMER_FLAG[9]
      ;ENDFOLD
      ;FOLD -- Warte Fraesen fertig oder Timeout -- ;%{SE}%MKUKATPVW %CVW_COM %VCOMMENT %P 2:-- Warte Fraesen fertig oder Timeout --, 3: VW_COMMENT
      ;ENDFOLD
      ;FOLD Schritt 260 = (F190 + T7 + T9 + F325) & A4039 ;%{SE}%MKUKATPVW %CVW_SPS %VST_CON %P 2:Schritt 260 = (F190 + T7 + T9 + F325) & A4039, 3: ST_CON
         IF ($FLAG[190] OR $TIMER_FLAG[7] OR $TIMER_FLAG[9] OR $FLAG[325]) AND $OUT[4039] THEN
            PREVSTEP = $APP_INT[5]
            $APP_INT[5] = 260
         ENDIF
      ;ENDFOLD
   ;ENDFOLD
   ;FOLD SCHRITT 260 -- MB1 Fraesen mit KFB1-- ;%{P}%MKUKATPVW,%CSTEP,%VST_NR,%P 1:SCHRITT, 2:260, 3: MB1 Fraesen mit KFB1
      ;FOLD ;%{H}
         Case 260
      ;ENDFOLD
      ;FOLD t9 ( EIN ) = STOP ;%{SE}%MKUKATPVW %CVW_SPS %VTSTOP %P 2:t9 ( EIN ) = STOP, 3: TSTOP
         VW(#SET_TIME,TRUE,9,1,0)
      ;ENDFOLD
      ;FOLD -- MB1 oeffnen -- ;%{SE}%MKUKATPVW %CVW_COM %VCOMMENT %P 2:-- MB1 oeffnen --, 3: VW_COMMENT
      ;ENDFOLD
      ;FOLD A1802 = AUS ;%{SE}%MKUKATPVW %CVW_SPS %VBOASG %P 2:A1802 = AUS, 3: BOASG
         $OUT[1802] = FALSE
      ;ENDFOLD
      ;FOLD A1798 = EIN ;%{SE}%MKUKATPVW %CVW_SPS %VBOASG %P 2:A1798 = EIN, 3: BOASG
         $OUT[1798] = TRUE
      ;ENDFOLD
      ;FOLD -- RSK Sammelstoerung -- ;%{SE}%MKUKATPVW %CVW_COM %VCOMMENT %P 2:-- RSK Sammelstoerung --, 3: VW_COMMENT
      ;ENDFOLD
      ;FOLD F329 = T7 + T9 + F325 ;%{SE}%MKUKATPVW %CVW_SPS %VBOASG %P 2:F329 = T7 + T9 + F325, 3: BOASG
         $FLAG[329] = $TIMER_FLAG[7] OR $TIMER_FLAG[9] OR $FLAG[325]
      ;ENDFOLD
      ;FOLD -- Weiter wenn Fraesen fertig -- ;%{SE}%MKUKATPVW %CVW_COM %VCOMMENT %P 2:-- Weiter wenn Fraesen fertig --, 3: VW_COMMENT
      ;ENDFOLD
      ;FOLD Schritt 261 = (E1798 & !E1802 & F190 + F325 + F329) & A4039 ;%{SE}%MKUKATPVW %CVW_SPS %VST_CON %P 2:Schritt 261 = (E1798 & !E1802 & F190 + F325 + F329) & A4039, 3: ST_CON
         IF ($IN[1798] AND NOT $IN[1802] AND $FLAG[190] OR $FLAG[325] OR $FLAG[329]) AND $OUT[4039] THEN
            PREVSTEP = $APP_INT[5]
            $APP_INT[5] = 261
         ENDIF
      ;ENDFOLD
   ;ENDFOLD
   ;FOLD SCHRITT 261 -- MB1 Fraesen mit KFB1 -- ;%{P}%MKUKATPVW,%CSTEP,%VST_NR,%P 1:SCHRITT, 2:261, 3: MB1 Fraesen mit KFB1
      ;FOLD ;%{H}
         Case 261
      ;ENDFOLD
      ;FOLD F324 = AUS ;%{SE}%MKUKATPVW %CVW_SPS %VBOASG %P 2:F324 = AUS, 3: BOASG
         $FLAG[324] = FALSE
      ;ENDFOLD
      ;FOLD A1798 = AUS ;%{SE}%MKUKATPVW %CVW_SPS %VBOASG %P 2:A1798 = AUS, 3: BOASG
         $OUT[1798] = FALSE
      ;ENDFOLD
      ;FOLD -- KFB1 abschalten -- ;%{SE}%MKUKATPVW %CVW_COM %VCOMMENT %P 2:-- KFB1 abschalten --, 3: VW_COMMENT
      ;ENDFOLD
      ;FOLD A1154 = AUS ;%{SE}%MKUKATPVW %CVW_SPS %VBOASG %P 2:A1154 = AUS, 3: BOASG
         $OUT[1154] = FALSE
      ;ENDFOLD
      ;FOLD -- Ueberwachungszeit KFB1 Versetzeinheit -- ;%{SE}%MKUKATPVW %CVW_COM %VCOMMENT %P 2:-- Ueberwachungszeit KFB1 Versetzeinheit --, 3: VW_COMMENT
      ;ENDFOLD
      ;FOLD t8 ( EIN ) = -20[1/10Sek] ;%{SE}%MKUKATPVW %CVW_SPS %VTASG %P 2:t8 ( EIN ) = -20[1/10Sek], 3: TASG
         VW(#SET_TIME,TRUE,8,0,-20)
      ;ENDFOLD
      ;FOLD Schritt 262 = A4039 ;%{SE}%MKUKATPVW %CVW_SPS %VST_CON %P 2:Schritt 262 = A4039, 3: ST_CON
         IF $OUT[4039] THEN
            PREVSTEP = $APP_INT[5]
            $APP_INT[5] = 262
         ENDIF
      ;ENDFOLD
   ;ENDFOLD
   ;FOLD SCHRITT 262 -- MB1 Fraesen mit KFB1 -- ;%{P}%MKUKATPVW,%CSTEP,%VST_NR,%P 1:SCHRITT, 2:262, 3: MB1 Fraesen mit KFB1
      ;FOLD ;%{H}
         Case 262
      ;ENDFOLD
      ;FOLD F328 = AUS ;%{SE}%MKUKATPVW %CVW_SPS %VBOASG %P 2:F328 = AUS, 3: BOASG
         $FLAG[328] = FALSE
      ;ENDFOLD
      ;FOLD -- KFB1 Versetzeinheit vor -- ;%{SE}%MKUKATPVW %CVW_COM %VCOMMENT %P 2:-- KFB1 Versetzeinheit vor --, 3: VW_COMMENT
      ;ENDFOLD
      ;FOLD A1155 = F564 ;%{SE}%MKUKATPVW %CVW_SPS %VBOASG %P 2:A1155 = F564, 3: BOASG
         $OUT[1155] = $FLAG[564]
      ;ENDFOLD
      ;FOLD -- RSK Fehlerausgabe KSB1 Arbeitsst. -- ;%{SE}%MKUKATPVW %CVW_COM %VCOMMENT %P 2:-- RSK Fehlerausgabe KSB1 Arbeitsst. --, 3: VW_COMMENT
      ;ENDFOLD
      ;FOLD F324 = !E1157 & !F323 & !F328 + F324 ;%{SE}%MKUKATPVW %CVW_SPS %VBOASG %P 2:F324 = !E1157 & !F323 & !F328 + F324, 3: BOASG
         $FLAG[324] = NOT $IN[1157] AND NOT $FLAG[323] AND NOT $FLAG[328] OR $FLAG[324]
      ;ENDFOLD
      ;FOLD -- RSK Sammelstoerung -- ;%{SE}%MKUKATPVW %CVW_COM %VCOMMENT %P 2:-- RSK Sammelstoerung --, 3: VW_COMMENT
      ;ENDFOLD
      ;FOLD F329 = F324 + F325 ;%{SE}%MKUKATPVW %CVW_SPS %VBOASG %P 2:F329 = F324 + F325, 3: BOASG
         $FLAG[329] = $FLAG[324] OR $FLAG[325]
      ;ENDFOLD
      ;FOLD Schritt 261 = F324 & (E26 + E27) & A4039 ;%{SE}%MKUKATPVW %CVW_SPS %VST_CON %P 2:Schritt 261 = F324 & (E26 + E27) & A4039, 3: ST_CON
         IF $FLAG[324] AND ($IN[26] OR $IN[27]) AND $OUT[4039] THEN
            PREVSTEP = $APP_INT[5]
            $APP_INT[5] = 261
         ENDIF
      ;ENDFOLD
      ;FOLD Schritt 263 = (!F324 & (E1155 & F564 + !E1155 & !F564) + T8 + F325) & A4039 ;%{SE}%MKUKATPVW %CVW_SPS %VST_CON %P 2:Schritt 263 = (!F324 & (E1155 & F564 + !E1155 & !F564) + T8 + F325) & A4039, 3: ST_CON
         IF (NOT $FLAG[324] AND ($IN[1155] AND $FLAG[564] OR NOT $IN[1155] AND NOT $FLAG[564]) OR $TIMER_FLAG[8] OR $FLAG[325]) AND $OUT[4039] THEN
            PREVSTEP = $APP_INT[5]
            $APP_INT[5] = 263
         ENDIF
      ;ENDFOLD
   ;ENDFOLD
   ;FOLD SCHRITT 263 -- MB1 Fraesen mit KFB1-- ;%{P}%MKUKATPVW,%CSTEP,%VST_NR,%P 1:SCHRITT, 2:263, 3: MB1 Fraesen mit KFB1
      ;FOLD ;%{H}
         Case 263
      ;ENDFOLD
      ;FOLD F323 = AUS ;%{SE}%MKUKATPVW %CVW_SPS %VBOASG %P 2:F323 = AUS, 3: BOASG
         $FLAG[323] = FALSE
      ;ENDFOLD
      ;FOLD F328 = AUS ;%{SE}%MKUKATPVW %CVW_SPS %VBOASG %P 2:F328 = AUS, 3: BOASG
         $FLAG[328] = FALSE
      ;ENDFOLD
      ;FOLD -- RSK Sammelstoerung -- ;%{SE}%MKUKATPVW %CVW_COM %VCOMMENT %P 2:-- RSK Sammelstoerung --, 3: VW_COMMENT
      ;ENDFOLD
      ;FOLD F329 = F325 ;%{SE}%MKUKATPVW %CVW_SPS %VBOASG %P 2:F329 = F325, 3: BOASG
         $FLAG[329] = $FLAG[325]
      ;ENDFOLD
      ;FOLD -- Ueberwachungszeit KSB1 schwenken -- ;%{SE}%MKUKATPVW %CVW_COM %VCOMMENT %P 2:-- Ueberwachungszeit KSB1 schwenken --, 3: VW_COMMENT
      ;ENDFOLD
      ;FOLD t8 ( EIN ) = -100[1/10Sek] ;%{SE}%MKUKATPVW %CVW_SPS %VTASG %P 2:t8 ( EIN ) = -100[1/10Sek], 3: TASG
         VW(#SET_TIME,TRUE,8,0,-100)
      ;ENDFOLD
      ;FOLD -- KFB1 Ausblasen ein -- ;%{SE}%MKUKATPVW %CVW_COM %VCOMMENT %P 2:-- KFB1 Ausblasen ein --, 3: VW_COMMENT
      ;ENDFOLD
      ;FOLD A1154 = EIN ;%{SE}%MKUKATPVW %CVW_SPS %VBOASG %P 2:A1154 = EIN, 3: BOASG
         $OUT[1154] = TRUE
      ;ENDFOLD
      ;FOLD -- KSB1 in Ruhestellung schwenken -- ;%{SE}%MKUKATPVW %CVW_COM %VCOMMENT %P 2:-- KSB1 in Ruhestellung schwenken --, 3: VW_COMMENT
      ;ENDFOLD
      ;FOLD A1160 = E1798 & (E1155 & F564 + !E1155 & !F564) ;%{SE}%MKUKATPVW %CVW_SPS %VBOASG %P 2:A1160 = E1798 & (E1155 & F564 + !E1155 & !F564), 3: BOASG
         $OUT[1160] = $IN[1798] AND ($IN[1155] AND $FLAG[564] OR NOT $IN[1155] AND NOT $FLAG[564])
      ;ENDFOLD
      ;FOLD Schritt 264 = E1798 & A1160 & A4039 ;%{SE}%MKUKATPVW %CVW_SPS %VST_CON %P 2:Schritt 264 = E1798 & A1160 & A4039, 3: ST_CON
         IF $IN[1798] AND $OUT[1160] AND $OUT[4039] THEN
            PREVSTEP = $APP_INT[5]
            $APP_INT[5] = 264
         ENDIF
      ;ENDFOLD
   ;ENDFOLD
   ;FOLD SCHRITT 264 -- MB1 Fraesen mit KFB1-- ;%{P}%MKUKATPVW,%CSTEP,%VST_NR,%P 1:SCHRITT, 2:264, 3: MB1 Fraesen mit KFB1
      ;FOLD ;%{H}
         Case 264
      ;ENDFOLD
      ;FOLD -- Hilfsflag SK Programmwechsel -- ;%{SE}%MKUKATPVW %CVW_COM %VCOMMENT %P 2:-- Hilfsflag SK Programmwechsel --, 3: VW_COMMENT
      ;ENDFOLD
      ;FOLD F334 = AUS ;%{SE}%MKUKATPVW %CVW_SPS %VBOASG %P 2:F334 = AUS, 3: BOASG
         $FLAG[334] = FALSE
      ;ENDFOLD
      ;FOLD -- RSK Fehlerausgabe KF Versetzeinheit -- ;%{SE}%MKUKATPVW %CVW_COM %VCOMMENT %P 2:-- RSK Fehlerausgabe KF Versetzeinheit --, 3: VW_COMMENT
      ;ENDFOLD
      ;FOLD F328 = !E1155 & F564 & !F323 + F328 ;%{SE}%MKUKATPVW %CVW_SPS %VBOASG %P 2:F328 = !E1155 & F564 & !F323 + F328, 3: BOASG
         $FLAG[328] = NOT $IN[1155] AND $FLAG[564] AND NOT $FLAG[323] OR $FLAG[328]
      ;ENDFOLD
      ;FOLD -- RSK Fehlerausgabe KSB1 Ruhestellung -- ;%{SE}%MKUKATPVW %CVW_COM %VCOMMENT %P 2:-- RSK Fehlerausgabe KSB1 Ruhestellung --, 3: VW_COMMENT
      ;ENDFOLD
      ;FOLD F323 = E1158 & T8 & (E1155 + !F564) + F323 ;%{SE}%MKUKATPVW %CVW_SPS %VBOASG %P 2:F323 = E1158 & T8 & (E1155 + !F564) + F323, 3: BOASG
         $FLAG[323] = $IN[1158] AND $TIMER_FLAG[8] AND ($IN[1155] OR NOT $FLAG[564]) OR $FLAG[323]
      ;ENDFOLD
      ;FOLD -- RSK Sammelstoerung -- ;%{SE}%MKUKATPVW %CVW_COM %VCOMMENT %P 2:-- RSK Sammelstoerung --, 3: VW_COMMENT
      ;ENDFOLD
      ;FOLD F329 = F323 + F325 + F328 ;%{SE}%MKUKATPVW %CVW_SPS %VBOASG %P 2:F329 = F323 + F325 + F328, 3: BOASG
         $FLAG[329] = $FLAG[323] OR $FLAG[325] OR $FLAG[328]
      ;ENDFOLD
      ;FOLD A1154 = !F323 & !F328 ;%{SE}%MKUKATPVW %CVW_SPS %VBOASG %P 2:A1154 = !F323 & !F328, 3: BOASG
         $OUT[1154] = NOT $FLAG[323] AND NOT $FLAG[328]
      ;ENDFOLD
      ;FOLD A1166 = !F323 & !F328 ;%{SE}%MKUKATPVW %CVW_SPS %VBOASG %P 2:A1166 = !F323 & !F328, 3: BOASG
         $OUT[1166] = NOT $FLAG[323] AND NOT $FLAG[328]
      ;ENDFOLD
      ;FOLD A1155 = !F323 & !F328 & F564 ;%{SE}%MKUKATPVW %CVW_SPS %VBOASG %P 2:A1155 = !F323 & !F328 & F564, 3: BOASG
         $OUT[1155] = NOT $FLAG[323] AND NOT $FLAG[328] AND $FLAG[564]
      ;ENDFOLD
      ;FOLD Schritt 262 = (F323 + F328) & (E26 + E27) & A4039 ;%{SE}%MKUKATPVW %CVW_SPS %VST_CON %P 2:Schritt 262 = (F323 + F328) & (E26 + E27) & A4039, 3: ST_CON
         IF ($FLAG[323] OR $FLAG[328]) AND ($IN[26] OR $IN[27]) AND $OUT[4039] THEN
            PREVSTEP = $APP_INT[5]
            $APP_INT[5] = 262
         ENDIF
      ;ENDFOLD
      ;FOLD Schritt 265 = E1156 & A4039 ;%{SE}%MKUKATPVW %CVW_SPS %VST_CON %P 2:Schritt 265 = E1156 & A4039, 3: ST_CON
         IF $IN[1156] AND $OUT[4039] THEN
            PREVSTEP = $APP_INT[5]
            $APP_INT[5] = 265
         ENDIF
      ;ENDFOLD
   ;ENDFOLD
   ;FOLD SCHRITT 265 -- MB1 Fraesen mit KFB1 -- ;%{P}%MKUKATPVW,%CSTEP,%VST_NR,%P 1:SCHRITT, 2:265, 3: MB1 Fraesen mit KFB1
      ;FOLD ;%{H}
         Case 265
      ;ENDFOLD
      ;FOLD F323 = AUS ;%{SE}%MKUKATPVW %CVW_SPS %VBOASG %P 2:F323 = AUS, 3: BOASG
         $FLAG[323] = FALSE
      ;ENDFOLD
      ;FOLD F328 = AUS ;%{SE}%MKUKATPVW %CVW_SPS %VBOASG %P 2:F328 = AUS, 3: BOASG
         $FLAG[328] = FALSE
      ;ENDFOLD
      ;FOLD -- RSK Sammelstoerung -- ;%{SE}%MKUKATPVW %CVW_COM %VCOMMENT %P 2:-- RSK Sammelstoerung --, 3: VW_COMMENT
      ;ENDFOLD
      ;FOLD F329 = F325 ;%{SE}%MKUKATPVW %CVW_SPS %VBOASG %P 2:F329 = F325, 3: BOASG
         $FLAG[329] = $FLAG[325]
      ;ENDFOLD
      ;FOLD t8 ( EIN ) = STOP ;%{SE}%MKUKATPVW %CVW_SPS %VTSTOP %P 2:t8 ( EIN ) = STOP, 3: TSTOP
         VW(#SET_TIME,TRUE,8,1,0)
      ;ENDFOLD
      ;FOLD -- KF1 Versetzeinheit rueck -- ;%{SE}%MKUKATPVW %CVW_COM %VCOMMENT %P 2:-- KF1 Versetzeinheit rueck --, 3: VW_COMMENT
      ;ENDFOLD
      ;FOLD A1155 = AUS ;%{SE}%MKUKATPVW %CVW_SPS %VBOASG %P 2:A1155 = AUS, 3: BOASG
         $OUT[1155] = FALSE
      ;ENDFOLD
      ;FOLD -- KFB1 Ausblasen aus -- ;%{SE}%MKUKATPVW %CVW_COM %VCOMMENT %P 2:-- KFB1 Ausblasen aus --, 3: VW_COMMENT
      ;ENDFOLD
      ;FOLD A1154 = AUS ;%{SE}%MKUKATPVW %CVW_SPS %VBOASG %P 2:A1154 = AUS, 3: BOASG
         $OUT[1154] = FALSE
      ;ENDFOLD
      ;FOLD A1166 = AUS ;%{SE}%MKUKATPVW %CVW_SPS %VBOASG %P 2:A1166 = AUS, 3: BOASG
         $OUT[1166] = FALSE
      ;ENDFOLD
      ;FOLD -- KSB1 in Ruhestellung schwenken AUS -- ;%{SE}%MKUKATPVW %CVW_COM %VCOMMENT %P 2:-- KSB1 in Ruhestellung schwenken AUS --, 3: VW_COMMENT
      ;ENDFOLD
      ;FOLD A1160 = AUS ;%{SE}%MKUKATPVW %CVW_SPS %VBOASG %P 2:A1160 = AUS, 3: BOASG
         $OUT[1160] = FALSE
      ;ENDFOLD
      ;FOLD -- Serviceprogramm Messen nach Fraesen an MB1 -- ;%{SE}%MKUKATPVW %CVW_COM %VCOMMENT %P 2:-- Serviceprogramm Messen nach Fraesen an MB1 --, 3: VW_COMMENT
      ;ENDFOLD
      ;FOLD bin7 ( !F329 ) = 25 ;%{SE}%MKUKATPVW %CVW_SPS %VARIASG %P 2:bin7 ( !F329 ) = 25, 3: ARIASG
         VW(#BINOUT,NOT $FLAG[329],7,25)
      ;ENDFOLD
      ;FOLD -- Wartezeit Programmwechsel SK -- ;%{SE}%MKUKATPVW %CVW_COM %VCOMMENT %P 2:-- Wartezeit Programmwechsel SK --, 3: VW_COMMENT
      ;ENDFOLD
      ;FOLD T8 ( !F334 ) = -2[1/10Sek] ;%{SE}%MKUKATPVW %CVW_SPS %VTASG %P 2:T8 ( !F334 ) = -2[1/10Sek], 3: TASG
         VW(#SET_TIME,NOT $FLAG[334],8,0,-2)
      ;ENDFOLD
      ;FOLD -- Hilfsflag SK Programmwechsel -- ;%{SE}%MKUKATPVW %CVW_COM %VCOMMENT %P 2:-- Hilfsflag SK Programmwechsel --, 3: VW_COMMENT
      ;ENDFOLD
      ;FOLD F334 = EIN ;%{SE}%MKUKATPVW %CVW_SPS %VBOASG %P 2:F334 = EIN, 3: BOASG
         $FLAG[334] = TRUE
      ;ENDFOLD
      ;FOLD -- Ueberwachungszeit MB1 Messen -- ;%{SE}%MKUKATPVW %CVW_COM %VCOMMENT %P 2:-- Ueberwachungszeit MB1 Messen --, 3: VW_COMMENT
      ;ENDFOLD
      ;FOLD t9 ( EIN ) = -100[1/10Sek] ;%{SE}%MKUKATPVW %CVW_SPS %VTASG %P 2:t9 ( EIN ) = -100[1/10Sek], 3: TASG
         VW(#SET_TIME,TRUE,9,0,-100)
      ;ENDFOLD
      ;FOLD Schritt 250 = (F325 + F329) & (E26 + E27) & A4039 ;%{SE}%MKUKATPVW %CVW_SPS %VST_CON %P 2:Schritt 250 = (F325 + F329) & (E26 + E27) & A4039, 3: ST_CON
         IF ($FLAG[325] OR $FLAG[329]) AND ($IN[26] OR $IN[27]) AND $OUT[4039] THEN
            PREVSTEP = $APP_INT[5]
            $APP_INT[5] = 250
         ENDIF
      ;ENDFOLD
      ;FOLD Schritt 266 = T8 & !F325 & !F329 & A4039 ;%{SE}%MKUKATPVW %CVW_SPS %VST_CON %P 2:Schritt 266 = T8 & !F325 & !F329 & A4039, 3: ST_CON
         IF $TIMER_FLAG[8] AND NOT $FLAG[325] AND NOT $FLAG[329] AND $OUT[4039] THEN
            PREVSTEP = $APP_INT[5]
            $APP_INT[5] = 266
         ENDIF
      ;ENDFOLD
   ;ENDFOLD
   ;FOLD SCHRITT 266 -- MB1 Fraesen mit KFB1 -- ;%{P}%MKUKATPVW,%CSTEP,%VST_NR,%P 1:SCHRITT, 2:266, 3: MB1 Fraesen mit KFB1
      ;FOLD ;%{H}
         Case 266
      ;ENDFOLD
      ;FOLD -- Hilfsflag SK Programmwechsel -- ;%{SE}%MKUKATPVW %CVW_COM %VCOMMENT %P 2:-- Hilfsflag SK Programmwechsel --, 3: VW_COMMENT
      ;ENDFOLD
      ;FOLD F334 = AUS ;%{SE}%MKUKATPVW %CVW_SPS %VBOASG %P 2:F334 = AUS, 3: BOASG
         $FLAG[334] = FALSE
      ;ENDFOLD
      ;FOLD -- RSK Sammelstoerung -- ;%{SE}%MKUKATPVW %CVW_COM %VCOMMENT %P 2:-- RSK Sammelstoerung --, 3: VW_COMMENT
      ;ENDFOLD
      ;FOLD F329 = T9 ;%{SE}%MKUKATPVW %CVW_SPS %VBOASG %P 2:F329 = T9, 3: BOASG
         $FLAG[329] = $TIMER_FLAG[9]
      ;ENDFOLD
      ;FOLD -- Messen nach Fraesen -- ;%{SE}%MKUKATPVW %CVW_COM %VCOMMENT %P 2:-- Messen nach Fraesen --, 3: VW_COMMENT
      ;ENDFOLD
      ;FOLD A1797 = !F329 ;%{SE}%MKUKATPVW %CVW_SPS %VBOASG %P 2:A1797 = !F329, 3: BOASG
         $OUT[1797] = NOT $FLAG[329]
      ;ENDFOLD
      ;FOLD Schritt 267 = E1818 & A4039 + T9 ;%{SE}%MKUKATPVW %CVW_SPS %VST_CON %P 2:Schritt 267 = E1818 & A4039 + T9, 3: ST_CON
         IF $IN[1818] AND $OUT[4039] OR $TIMER_FLAG[9] THEN
            PREVSTEP = $APP_INT[5]
            $APP_INT[5] = 267
         ENDIF
      ;ENDFOLD
   ;ENDFOLD
   ;FOLD SCHRITT 267 -- MB1 Fraesen mit KFB1 -- ;%{P}%MKUKATPVW,%CSTEP,%VST_NR,%P 1:SCHRITT, 2:267, 3: MB1 Fraesen mit KFB1
      ;FOLD ;%{H}
         Case 267
      ;ENDFOLD
      ;FOLD -- RSK Sammelstoerung -- ;%{SE}%MKUKATPVW %CVW_COM %VCOMMENT %P 2:-- RSK Sammelstoerung --, 3: VW_COMMENT
      ;ENDFOLD
      ;FOLD F329 = T9 ;%{SE}%MKUKATPVW %CVW_SPS %VBOASG %P 2:F329 = T9, 3: BOASG
         $FLAG[329] = $TIMER_FLAG[9]
      ;ENDFOLD
      ;FOLD A1797 = AUS ;%{SE}%MKUKATPVW %CVW_SPS %VBOASG %P 2:A1797 = AUS, 3: BOASG
         $OUT[1797] = FALSE
      ;ENDFOLD
      ;FOLD Schritt 268 = E1818 & A4039 + T9 ;%{SE}%MKUKATPVW %CVW_SPS %VST_CON %P 2:Schritt 268 = E1818 & A4039 + T9, 3: ST_CON
         IF $IN[1818] AND $OUT[4039] OR $TIMER_FLAG[9] THEN
            PREVSTEP = $APP_INT[5]
            $APP_INT[5] = 268
         ENDIF
      ;ENDFOLD
   ;ENDFOLD
   ;FOLD SCHRITT 268 -- MB1 Fraesen mit KFB1 -- ;%{P}%MKUKATPVW,%CSTEP,%VST_NR,%P 1:SCHRITT, 2:268, 3: MB1 Fraesen mit KFB1
      ;FOLD ;%{H}
         Case 268
      ;ENDFOLD
      ;FOLD -- Hilfsflag SK Programmwechsel -- ;%{SE}%MKUKATPVW %CVW_COM %VCOMMENT %P 2:-- Hilfsflag SK Programmwechsel --, 3: VW_COMMENT
      ;ENDFOLD
      ;FOLD F334 = AUS ;%{SE}%MKUKATPVW %CVW_SPS %VBOASG %P 2:F334 = AUS, 3: BOASG
         $FLAG[334] = FALSE
      ;ENDFOLD
      ;FOLD t9 ( EIN ) = STOP ;%{SE}%MKUKATPVW %CVW_SPS %VTSTOP %P 2:t9 ( EIN ) = STOP, 3: TSTOP
         VW(#SET_TIME,TRUE,9,1,0)
      ;ENDFOLD
      ;FOLD -- RSK Fehlerausgabe Messen -- ;%{SE}%MKUKATPVW %CVW_COM %VCOMMENT %P 2:-- RSK Fehlerausgabe Messen --, 3: VW_COMMENT
      ;ENDFOLD
      ;FOLD F327 = E1820 + T9 ;%{SE}%MKUKATPVW %CVW_SPS %VBOASG %P 2:F327 = E1820 + T9, 3: BOASG
         $FLAG[327] = $IN[1820] OR $TIMER_FLAG[9]
      ;ENDFOLD
      ;FOLD -- RSK Sammelstoerung -- ;%{SE}%MKUKATPVW %CVW_COM %VCOMMENT %P 2:-- RSK Sammelstoerung --, 3: VW_COMMENT
      ;ENDFOLD
      ;FOLD F329 = F327 ;%{SE}%MKUKATPVW %CVW_SPS %VBOASG %P 2:F329 = F327, 3: BOASG
         $FLAG[329] = $FLAG[327]
      ;ENDFOLD
      ;FOLD Schritt 250 = F329 & (E26 + E27) & A4039 ;%{SE}%MKUKATPVW %CVW_SPS %VST_CON %P 2:Schritt 250 = F329 & (E26 + E27) & A4039, 3: ST_CON
         IF $FLAG[329] AND ($IN[26] OR $IN[27]) AND $OUT[4039] THEN
            PREVSTEP = $APP_INT[5]
            $APP_INT[5] = 250
         ENDIF
      ;ENDFOLD
      ;FOLD Schritt 269 = !F329 & A4039 ;%{SE}%MKUKATPVW %CVW_SPS %VST_CON %P 2:Schritt 269 = !F329 & A4039, 3: ST_CON
         IF NOT $FLAG[329] AND $OUT[4039] THEN
            PREVSTEP = $APP_INT[5]
            $APP_INT[5] = 269
         ENDIF
      ;ENDFOLD
   ;ENDFOLD
   ;FOLD SCHRITT 269 -- MB1 Fraesen mit KFB1 -- ;%{P}%MKUKATPVW,%CSTEP,%VST_NR,%P 1:SCHRITT, 2:269, 3: MB1 Fraesen mit KFB1
      ;FOLD ;%{H}
         Case 269
      ;ENDFOLD
      ;FOLD bin7 ( !F326 ) = 1 ;%{SE}%MKUKATPVW %CVW_SPS %VARIASG %P 2:bin7 ( !F326 ) = 1, 3: ARIASG
         VW(#BINOUT,NOT $FLAG[326],7,1)
      ;ENDFOLD
      ;FOLD -- Wartezeit Programmwechsel SK -- ;%{SE}%MKUKATPVW %CVW_COM %VCOMMENT %P 2:-- Wartezeit Programmwechsel SK --, 3: VW_COMMENT
      ;ENDFOLD
      ;FOLD T8 ( !F334 ) = -2[1/10Sek] ;%{SE}%MKUKATPVW %CVW_SPS %VTASG %P 2:T8 ( !F334 ) = -2[1/10Sek], 3: TASG
         VW(#SET_TIME,NOT $FLAG[334],8,0,-2)
      ;ENDFOLD
      ;FOLD -- Hilfsflag SK Programmwechsel -- ;%{SE}%MKUKATPVW %CVW_COM %VCOMMENT %P 2:-- Hilfsflag SK Programmwechsel --, 3: VW_COMMENT
      ;ENDFOLD
      ;FOLD F334 = EIN ;%{SE}%MKUKATPVW %CVW_SPS %VBOASG %P 2:F334 = EIN, 3: BOASG
         $FLAG[334] = TRUE
      ;ENDFOLD
      ;FOLD t9 ( EIN ) = -40[1/10Sek] ;%{SE}%MKUKATPVW %CVW_SPS %VTASG %P 2:t9 ( EIN ) = -40[1/10Sek], 3: TASG
         VW(#SET_TIME,TRUE,9,0,-40)
      ;ENDFOLD
      ;FOLD Schritt 250 = E1820 & !E1819 & (F322 + F323 + F325 + F326 + F327 + F329) & (E26 + E27) & A4039 ;%{SE}%MKUKATPVW %CVW_SPS %VST_CON %P 2:Schritt 250 = E1820 & !E1819 & (F322 + F323 + F325 + F326 + F327 + F329) & (E26 + E27) & A4039, 3: ST_CON
         IF $IN[1820] AND NOT $IN[1819] AND ($FLAG[322] OR $FLAG[323] OR $FLAG[325] OR $FLAG[326] OR $FLAG[327] OR $FLAG[329]) AND ($IN[26] OR $IN[27]) AND $OUT[4039] THEN
            PREVSTEP = $APP_INT[5]
            $APP_INT[5] = 250
         ENDIF
      ;ENDFOLD
      ;FOLD Schritt 270 = T8 & !E1820 & E1819 & (!F325 & !F329 & !F326 & !F327) & A4039 ;%{SE}%MKUKATPVW %CVW_SPS %VST_CON %P 2:Schritt 270 = T8 & !E1820 & E1819 & (!F325 & !F329 & !F326 & !F327) & A4039, 3: ST_CON
         IF $TIMER_FLAG[8] AND NOT $IN[1820] AND $IN[1819] AND (NOT $FLAG[325] AND NOT $FLAG[329] AND NOT $FLAG[326] AND NOT $FLAG[327]) AND $OUT[4039] THEN
            PREVSTEP = $APP_INT[5]
            $APP_INT[5] = 270
         ENDIF
      ;ENDFOLD
   ;ENDFOLD
   ;FOLD SCHRITT 270 -- MB1 Fraesen mit KFB1-- ;%{P}%MKUKATPVW,%CSTEP,%VST_NR,%P 1:SCHRITT, 2:270, 3: MB1 Fraesen mit KFB1
      ;FOLD ;%{H}
         Case 270
      ;ENDFOLD
      ;FOLD -- Hilfsflag SK Programmwechsel -- ;%{SE}%MKUKATPVW %CVW_COM %VCOMMENT %P 2:-- Hilfsflag SK Programmwechsel --, 3: VW_COMMENT
      ;ENDFOLD
      ;FOLD F334 = AUS ;%{SE}%MKUKATPVW %CVW_SPS %VBOASG %P 2:F334 = AUS, 3: BOASG
         $FLAG[334] = FALSE
      ;ENDFOLD
      ;FOLD -- Quittierung Fraesen -- ;%{SE}%MKUKATPVW %CVW_COM %VCOMMENT %P 2:-- Quittierung Fraesen --, 3: VW_COMMENT
      ;ENDFOLD
      ;FOLD A1813 = E1819 ;%{SE}%MKUKATPVW %CVW_SPS %VBOASG %P 2:A1813 = E1819, 3: BOASG
         $OUT[1813] = $IN[1819]
      ;ENDFOLD
      ;FOLD Schritt 271 = !E1812 & A4039 ;%{SE}%MKUKATPVW %CVW_SPS %VST_CON %P 2:Schritt 271 = !E1812 & A4039, 3: ST_CON
         IF NOT $IN[1812] AND $OUT[4039] THEN
            PREVSTEP = $APP_INT[5]
            $APP_INT[5] = 271
         ENDIF
      ;ENDFOLD
   ;ENDFOLD
   ;FOLD SCHRITT 271 -- MB1 Fraesen mit KFB1 # Ende -- ;%{P}%MKUKATPVW,%CSTEP,%VST_NR,%P 1:SCHRITT, 2:271, 3: MB1 Fraesen mit KFB1 # Ende
      ;FOLD ;%{H}
         Case 271
      ;ENDFOLD
      ;FOLD -- RSK Sammelstoerung -- ;%{SE}%MKUKATPVW %CVW_COM %VCOMMENT %P 2:-- RSK Sammelstoerung --, 3: VW_COMMENT
      ;ENDFOLD
      ;FOLD F329 = T9 ;%{SE}%MKUKATPVW %CVW_SPS %VBOASG %P 2:F329 = T9, 3: BOASG
         $FLAG[329] = $TIMER_FLAG[9]
      ;ENDFOLD
      ;FOLD A1813 = AUS ;%{SE}%MKUKATPVW %CVW_SPS %VBOASG %P 2:A1813 = AUS, 3: BOASG
         $OUT[1813] = FALSE
      ;ENDFOLD
      ;FOLD A1812 = AUS ;%{SE}%MKUKATPVW %CVW_SPS %VBOASG %P 2:A1812 = AUS, 3: BOASG
         $OUT[1812] = FALSE
      ;ENDFOLD
      ;FOLD F210 = !E1812 ;%{SE}%MKUKATPVW %CVW_SPS %VBOASG %P 2:F210 = !E1812, 3: BOASG
         $FLAG[210] = NOT $IN[1812]
      ;ENDFOLD
      ;FOLD Schritt 1 = F210 & A4039 ;%{SE}%MKUKATPVW %CVW_SPS %VST_CON %P 2:Schritt 1 = F210 & A4039, 3: ST_CON
         IF $FLAG[210] AND $OUT[4039] THEN
            PREVSTEP = $APP_INT[5]
            $APP_INT[5] = 1
         ENDIF
      ;ENDFOLD
   ;ENDFOLD
   ;FOLD SCHRITT 272 -- ROB STP1 SZ1 # Start-- ;%{P}%MKUKATPVW,%CSTEP,%VST_NR,%P 1:SCHRITT, 2:272, 3: ROB STP1 SZ1 # Start
      ;FOLD ;%{H}
         Case 272
      ;ENDFOLD
      ;FOLD -- RSK gestartet -- ;%{SE}%MKUKATPVW %CVW_COM %VCOMMENT %P 2:-- RSK gestartet --, 3: VW_COMMENT
      ;ENDFOLD
      ;FOLD F321 = AUS ;%{SE}%MKUKATPVW %CVW_SPS %VBOASG %P 2:F321 = AUS, 3: BOASG
         $FLAG[321] = FALSE
      ;ENDFOLD
      ;FOLD F322 = AUS ;%{SE}%MKUKATPVW %CVW_SPS %VBOASG %P 2:F322 = AUS, 3: BOASG
         $FLAG[322] = FALSE
      ;ENDFOLD
      ;FOLD F323 = AUS ;%{SE}%MKUKATPVW %CVW_SPS %VBOASG %P 2:F323 = AUS, 3: BOASG
         $FLAG[323] = FALSE
      ;ENDFOLD
      ;FOLD F324 = AUS ;%{SE}%MKUKATPVW %CVW_SPS %VBOASG %P 2:F324 = AUS, 3: BOASG
         $FLAG[324] = FALSE
      ;ENDFOLD
      ;FOLD F325 = AUS ;%{SE}%MKUKATPVW %CVW_SPS %VBOASG %P 2:F325 = AUS, 3: BOASG
         $FLAG[325] = FALSE
      ;ENDFOLD
      ;FOLD F327 = AUS ;%{SE}%MKUKATPVW %CVW_SPS %VBOASG %P 2:F327 = AUS, 3: BOASG
         $FLAG[327] = FALSE
      ;ENDFOLD
      ;FOLD F329 = AUS ;%{SE}%MKUKATPVW %CVW_SPS %VBOASG %P 2:F329 = AUS, 3: BOASG
         $FLAG[329] = FALSE
      ;ENDFOLD
      ;FOLD -- EZ1/SP1/KE1 SZ1 Zaehler -- ;%{SE}%MKUKATPVW %CVW_COM %VCOMMENT %P 2:-- EZ1/SP1/KE1 SZ1 Zaehler --, 3: VW_COMMENT
      ;ENDFOLD
      ;FOLD F94 = AUS ;%{SE}%MKUKATPVW %CVW_SPS %VBOASG %P 2:F94 = AUS, 3: BOASG
         $FLAG[94] = FALSE
      ;ENDFOLD
      ;FOLD F95 = AUS ;%{SE}%MKUKATPVW %CVW_SPS %VBOASG %P 2:F95 = AUS, 3: BOASG
         $FLAG[95] = FALSE
      ;ENDFOLD
      ;FOLD F96 = AUS ;%{SE}%MKUKATPVW %CVW_SPS %VBOASG %P 2:F96 = AUS, 3: BOASG
         $FLAG[96] = FALSE
      ;ENDFOLD
      ;FOLD F97 = AUS ;%{SE}%MKUKATPVW %CVW_SPS %VBOASG %P 2:F97 = AUS, 3: BOASG
         $FLAG[97] = FALSE
      ;ENDFOLD
      ;FOLD F98 = AUS ;%{SE}%MKUKATPVW %CVW_SPS %VBOASG %P 2:F98 = AUS, 3: BOASG
         $FLAG[98] = FALSE
      ;ENDFOLD
      ;FOLD F99 = AUS ;%{SE}%MKUKATPVW %CVW_SPS %VBOASG %P 2:F99 = AUS, 3: BOASG
         $FLAG[99] = FALSE
      ;ENDFOLD
      ;FOLD -- Hilfsflags Funktionstest KF Motor -- ;%{SE}%MKUKATPVW %CVW_COM %VCOMMENT %P 2:-- Hilfsflags Funktionstest KF Motor --, 3: VW_COMMENT
      ;ENDFOLD
      ;FOLD F312 = AUS ;%{SE}%MKUKATPVW %CVW_SPS %VBOASG %P 2:F312 = AUS, 3: BOASG
         $FLAG[312] = FALSE
      ;ENDFOLD
      ;FOLD F313 = AUS ;%{SE}%MKUKATPVW %CVW_SPS %VBOASG %P 2:F313 = AUS, 3: BOASG
         $FLAG[313] = FALSE
      ;ENDFOLD
      ;FOLD -- Ueberwachungszeit KF1 -- ;%{SE}%MKUKATPVW %CVW_COM %VCOMMENT %P 2:-- Ueberwachungszeit KF1 --, 3: VW_COMMENT
      ;ENDFOLD
      ;FOLD t7 ( EIN ) = -30[1/10Sek] ;%{SE}%MKUKATPVW %CVW_SPS %VTASG %P 2:t7 ( EIN ) = -30[1/10Sek], 3: TASG
         VW(#SET_TIME,TRUE,7,0,-30)
      ;ENDFOLD
      ;FOLD Schritt 273 = A4039 ;%{SE}%MKUKATPVW %CVW_SPS %VST_CON %P 2:Schritt 273 = A4039, 3: ST_CON
         IF $OUT[4039] THEN
            PREVSTEP = $APP_INT[5]
            $APP_INT[5] = 273
         ENDIF
      ;ENDFOLD
   ;ENDFOLD
   ;FOLD SCHRITT 273 -- ROB STP1 SZ1-- ;%{P}%MKUKATPVW,%CSTEP,%VST_NR,%P 1:SCHRITT, 2:273, 3: ROB STP1 SZ1
      ;FOLD ;%{H}
         Case 273
      ;ENDFOLD
      ;FOLD i1 (EIN) = 0 ;%{SE}%MKUKATPVW %CVW_SPS %VARIASG %P 2:i1 (EIN) = 0, 3: ARIASG
         VW(#COUNTER,TRUE,1,0)
      ;ENDFOLD
      ;FOLD A858 = F537 ;%{SE}%MKUKATPVW %CVW_SPS %VBOASG %P 2:A858 = F537, 3: BOASG
         $OUT[858] = $FLAG[537]
      ;ENDFOLD
      ;FOLD A860 = F537 ;%{SE}%MKUKATPVW %CVW_SPS %VBOASG %P 2:A860 = F537, 3: BOASG
         $OUT[860] = $FLAG[537]
      ;ENDFOLD
      ;FOLD A834 = !F537 ;%{SE}%MKUKATPVW %CVW_SPS %VBOASG %P 2:A834 = !F537, 3: BOASG
         $OUT[834] = NOT $FLAG[537]
      ;ENDFOLD
      ;FOLD Schritt 274 = A4039 ;%{SE}%MKUKATPVW %CVW_SPS %VST_CON %P 2:Schritt 274 = A4039, 3: ST_CON
         IF $OUT[4039] THEN
            PREVSTEP = $APP_INT[5]
            $APP_INT[5] = 274
         ENDIF
      ;ENDFOLD
   ;ENDFOLD
   ;FOLD SCHRITT 274 -- ROB STP1 SZ1-- ;%{P}%MKUKATPVW,%CSTEP,%VST_NR,%P 1:SCHRITT, 2:274, 3: ROB STP1 SZ1
      ;FOLD ;%{H}
         Case 274
      ;ENDFOLD
      ;FOLD -- Funktionstest KF Motor -- ;%{SE}%MKUKATPVW %CVW_COM %VCOMMENT %P 2:-- Funktionstest KF Motor --, 3: VW_COMMENT
      ;ENDFOLD
      ;FOLD F312 = EIN ;%{SE}%MKUKATPVW %CVW_SPS %VBOASG %P 2:F312 = EIN, 3: BOASG
         $FLAG[312] = TRUE
      ;ENDFOLD
      ;FOLD F313 = i1 > 2 ;%{SE}%MKUKATPVW %CVW_SPS %VBOCMP %P 2:F313 = i1 > 2, 3: BOCMP
         $FLAG[313] = $COUNT_I[1] > 2
      ;ENDFOLD
      ;FOLD Schritt 275 = (F313 + T7) & A4039 ;%{SE}%MKUKATPVW %CVW_SPS %VST_CON %P 2:Schritt 275 = (F313 + T7) & A4039, 3: ST_CON
         IF ($FLAG[313] OR $TIMER_FLAG[7]) AND $OUT[4039] THEN
            PREVSTEP = $APP_INT[5]
            $APP_INT[5] = 275
         ENDIF
      ;ENDFOLD
   ;ENDFOLD
   ;FOLD SCHRITT 275 -- ROB STP1 SZ1-- ;%{P}%MKUKATPVW,%CSTEP,%VST_NR,%P 1:SCHRITT, 2:275, 3: ROB STP1 SZ1
      ;FOLD ;%{H}
         Case 275
      ;ENDFOLD
      ;FOLD F312 = AUS ;%{SE}%MKUKATPVW %CVW_SPS %VBOASG %P 2:F312 = AUS, 3: BOASG
         $FLAG[312] = FALSE
      ;ENDFOLD
      ;FOLD -- RSK Fehlerausgabe KF1 Initiator/Motor -- ;%{SE}%MKUKATPVW %CVW_COM %VCOMMENT %P 2:-- RSK Fehlerausgabe KF1 Initiator/Motor --, 3: VW_COMMENT
      ;ENDFOLD
      ;FOLD F322 = !F313 ;%{SE}%MKUKATPVW %CVW_SPS %VBOASG %P 2:F322 = !F313, 3: BOASG
         $FLAG[322] = NOT $FLAG[313]
      ;ENDFOLD
      ;FOLD -- RSK Sammelstoerung -- ;%{SE}%MKUKATPVW %CVW_COM %VCOMMENT %P 2:-- RSK Sammelstoerung --, 3: VW_COMMENT
      ;ENDFOLD
      ;FOLD F329 = F322 ;%{SE}%MKUKATPVW %CVW_SPS %VBOASG %P 2:F329 = F322, 3: BOASG
         $FLAG[329] = $FLAG[322]
      ;ENDFOLD
      ;FOLD T7 ( EIN ) = STOP ;%{SE}%MKUKATPVW %CVW_SPS %VTSTOP %P 2:T7 ( EIN ) = STOP, 3: TSTOP
         VW(#SET_TIME,TRUE,7,1,0)
      ;ENDFOLD
      ;FOLD A834 = !F322 & !F537 ;%{SE}%MKUKATPVW %CVW_SPS %VBOASG %P 2:A834 = !F322 & !F537, 3: BOASG
         $OUT[834] = NOT $FLAG[322] AND NOT $FLAG[537]
      ;ENDFOLD
      ;FOLD A858 = !F322 & F537 ;%{SE}%MKUKATPVW %CVW_SPS %VBOASG %P 2:A858 = !F322 & F537, 3: BOASG
         $OUT[858] = NOT $FLAG[322] AND $FLAG[537]
      ;ENDFOLD
      ;FOLD A860 = A858 ;%{SE}%MKUKATPVW %CVW_SPS %VBOASG %P 2:A860 = A858, 3: BOASG
         $OUT[860] = $OUT[858]
      ;ENDFOLD
      ;FOLD Schritt 276 = !F322 & A4039 ;%{SE}%MKUKATPVW %CVW_SPS %VST_CON %P 2:Schritt 276 = !F322 & A4039, 3: ST_CON
         IF NOT $FLAG[322] AND $OUT[4039] THEN
            PREVSTEP = $APP_INT[5]
            $APP_INT[5] = 276
         ENDIF
      ;ENDFOLD
      ;FOLD Schritt 278 = F322 & A4039 ;%{SE}%MKUKATPVW %CVW_SPS %VST_CON %P 2:Schritt 278 = F322 & A4039, 3: ST_CON
         IF $FLAG[322] AND $OUT[4039] THEN
            PREVSTEP = $APP_INT[5]
            $APP_INT[5] = 278
         ENDIF
      ;ENDFOLD
   ;ENDFOLD
   ;FOLD SCHRITT 276 -- ROB STP1 SZ1-- ;%{P}%MKUKATPVW,%CSTEP,%VST_NR,%P 1:SCHRITT, 2:276, 3: ROB STP1 SZ1
      ;FOLD ;%{H}
         Case 276
      ;ENDFOLD
      ;FOLD F312 = AUS ;%{SE}%MKUKATPVW %CVW_SPS %VBOASG %P 2:F312 = AUS, 3: BOASG
         $FLAG[312] = FALSE
      ;ENDFOLD
      ;FOLD F313 = AUS ;%{SE}%MKUKATPVW %CVW_SPS %VBOASG %P 2:F313 = AUS, 3: BOASG
         $FLAG[313] = FALSE
      ;ENDFOLD
      ;FOLD -- Umdreh. KF setzen zwischenspeichern -- ;%{SE}%MKUKATPVW %CVW_COM %VCOMMENT %P 2:-- Umdreh. KF setzen zwischenspeichern --, 3: VW_COMMENT
      ;ENDFOLD
      ;FOLD i45 ( EIN ) = i4 ;%{SE}%MKUKATPVW %CVW_SPS %VARIASG %P 2:i45 ( EIN ) = i4, 3: ARIASG
         VW(#COUNTER,TRUE,45,$COUNT_I[4])
      ;ENDFOLD
      ;FOLD i4 ( F99 ) = i33 ;%{SE}%MKUKATPVW %CVW_SPS %VARIASG %P 2:i4 ( F99 ) = i33, 3: ARIASG
         VW(#COUNTER,$FLAG[99],4,$COUNT_I[33])
      ;ENDFOLD
      ;FOLD i1 ( EIN ) = 0 ;%{SE}%MKUKATPVW %CVW_SPS %VARIASG %P 2:i1 ( EIN ) = 0, 3: ARIASG
         VW(#COUNTER,TRUE,1,0)
      ;ENDFOLD
      ;FOLD -- Ueberwachungszeit EZ1/SP1/KE1 SZ1 schliessen -- ;%{SE}%MKUKATPVW %CVW_COM %VCOMMENT %P 2:-- Ueberwachungszeit EZ1/SP1/KE1 SZ1 schliessen --, 3: VW_COMMENT
      ;ENDFOLD
      ;FOLD t9 ( EIN ) = -40[1/10Sek] ;%{SE}%MKUKATPVW %CVW_SPS %VTASG %P 2:t9 ( EIN ) = -40[1/10Sek], 3: TASG
         VW(#SET_TIME,TRUE,9,0,-40)
      ;ENDFOLD
      ;FOLD -- Ueberwachungszeit KF1 -- ;%{SE}%MKUKATPVW %CVW_COM %VCOMMENT %P 2:-- Ueberwachungszeit KF1 --, 3: VW_COMMENT
      ;ENDFOLD
      ;FOLD t7 ( EIN ) = -40[1/10Sek] ;%{SE}%MKUKATPVW %CVW_SPS %VTASG %P 2:t7 ( EIN ) = -40[1/10Sek], 3: TASG
         VW(#SET_TIME,TRUE,7,0,-40)
      ;ENDFOLD
      ;FOLD -- Wiederholung beim Startfraesen -- ;%{SE}%MKUKATPVW %CVW_COM %VCOMMENT %P 2:-- Wiederholung beim Startfraesen --, 3: VW_COMMENT
      ;ENDFOLD
      ;FOLD Schritt 277 = A4039 ;%{SE}%MKUKATPVW %CVW_SPS %VST_CON %P 2:Schritt 277 = A4039, 3: ST_CON
         IF $OUT[4039] THEN
            PREVSTEP = $APP_INT[5]
            $APP_INT[5] = 277
         ENDIF
      ;ENDFOLD
   ;ENDFOLD
   ;FOLD SCHRITT 277 -- ROB STP1 SZ1-- ;%{P}%MKUKATPVW,%CSTEP,%VST_NR,%P 1:SCHRITT, 2:277, 3: ROB STP1 SZ1
      ;FOLD ;%{H}
         Case 277
      ;ENDFOLD
      ;FOLD -- KF1 Ausblasen -- ;%{SE}%MKUKATPVW %CVW_COM %VCOMMENT %P 2:-- KF1 Ausblasen --, 3: VW_COMMENT
      ;ENDFOLD
      ;FOLD A836 = AUS ;%{SE}%MKUKATPVW %CVW_SPS %VBOASG %P 2:A836 = AUS, 3: BOASG
         $OUT[836] = FALSE
      ;ENDFOLD
      ;FOLD A860 = A836 ;%{SE}%MKUKATPVW %CVW_SPS %VBOASG %P 2:A860 = A836, 3: BOASG
         $OUT[860] = $OUT[836]
      ;ENDFOLD
      ;FOLD Schritt 278 = E858 & A4039 ;%{SE}%MKUKATPVW %CVW_SPS %VST_CON %P 2:Schritt 278 = E858 & A4039, 3: ST_CON
         IF $IN[858] AND $OUT[4039] THEN
            PREVSTEP = $APP_INT[5]
            $APP_INT[5] = 278
         ENDIF
      ;ENDFOLD
   ;ENDFOLD
   ;FOLD SCHRITT 278 -- ROB STP1 SZ1-- ;%{P}%MKUKATPVW,%CSTEP,%VST_NR,%P 1:SCHRITT, 2:278, 3: ROB STP1 SZ1
      ;FOLD ;%{H}
         Case 278
      ;ENDFOLD
      ;FOLD -- EZ1/SP1/KE1 SZ1 schliessen -- ;%{SE}%MKUKATPVW %CVW_COM %VCOMMENT %P 2:-- EZ1/SP1/KE1 SZ1 schliessen --, 3: VW_COMMENT
      ;ENDFOLD
      ;FOLD A717 = AUS ;%{SE}%MKUKATPVW %CVW_SPS %VBOASG %P 2:A717 = AUS, 3: BOASG
         $OUT[717] = FALSE
      ;ENDFOLD
      ;FOLD A720 = EIN ;%{SE}%MKUKATPVW %CVW_SPS %VBOASG %P 2:A720 = EIN, 3: BOASG
         $OUT[720] = TRUE
      ;ENDFOLD
      ;FOLD A718 = EIN ;%{SE}%MKUKATPVW %CVW_SPS %VBOASG %P 2:A718 = EIN, 3: BOASG
         $OUT[718] = TRUE
      ;ENDFOLD
      ;FOLD t11 ( EIN ) = -5[1/10Sek] ;%{SE}%MKUKATPVW %CVW_SPS %VTASG %P 2:t11 ( EIN ) = -5[1/10Sek], 3: TASG
         VW(#SET_TIME,TRUE,11,0,-5)
      ;ENDFOLD
      ;FOLD A720 = T11 ;%{SE}%MKUKATPVW %CVW_SPS %VBOASG %P 2:A720 = T11, 3: BOASG
         $OUT[720] = $TIMER_FLAG[11]
      ;ENDFOLD
      ;FOLD -- Ueberwachungszeit KF1 -- ;%{SE}%MKUKATPVW %CVW_COM %VCOMMENT %P 2:-- Ueberwachungszeit KF1 --, 3: VW_COMMENT
      ;ENDFOLD
      ;FOLD Schritt 279 = (E718 + T9) & A4039 ;%{SE}%MKUKATPVW %CVW_SPS %VST_CON %P 2:Schritt 279 = (E718 + T9) & A4039, 3: ST_CON
         IF ($IN[718] OR $TIMER_FLAG[9]) AND $OUT[4039] THEN
            PREVSTEP = $APP_INT[5]
            $APP_INT[5] = 279
         ENDIF
      ;ENDFOLD
   ;ENDFOLD
   ;FOLD SCHRITT 279 -- ROB STP1 SZ1 -- ;%{P}%MKUKATPVW,%CSTEP,%VST_NR,%P 1:SCHRITT, 2:279, 3: ROB STP1 SZ1
      ;FOLD ;%{H}
         Case 279
      ;ENDFOLD
      ;FOLD T9 ( EIN ) = STOP ;%{SE}%MKUKATPVW %CVW_SPS %VTSTOP %P 2:T9 ( EIN ) = STOP, 3: TSTOP
         VW(#SET_TIME,TRUE,9,1,0)
      ;ENDFOLD
      ;FOLD -- RSK Fehlerausgabe Kraftaufbau -- ;%{SE}%MKUKATPVW %CVW_COM %VCOMMENT %P 2:-- RSK Fehlerausgabe Kraftaufbau --, 3: VW_COMMENT
      ;ENDFOLD
      ;FOLD F325 = T9 ;%{SE}%MKUKATPVW %CVW_SPS %VBOASG %P 2:F325 = T9, 3: BOASG
         $FLAG[325] = $TIMER_FLAG[9]
      ;ENDFOLD
      ;FOLD -- KF1 abschalten bei Fehler -- ;%{SE}%MKUKATPVW %CVW_COM %VCOMMENT %P 2:-- KF1 abschalten bei Fehler --, 3: VW_COMMENT
      ;ENDFOLD
      ;FOLD A834 = !T7 & !T9 ;%{SE}%MKUKATPVW %CVW_SPS %VBOASG %P 2:A834 = !T7 & !T9, 3: BOASG
         $OUT[834] = NOT $TIMER_FLAG[7] AND NOT $TIMER_FLAG[9]
      ;ENDFOLD
      ;FOLD A858 = !T7 & !T9 ;%{SE}%MKUKATPVW %CVW_SPS %VBOASG %P 2:A858 = !T7 & !T9, 3: BOASG
         $OUT[858] = NOT $TIMER_FLAG[7] AND NOT $TIMER_FLAG[9]
      ;ENDFOLD
      ;FOLD A860 = !T7 & !T9 ;%{SE}%MKUKATPVW %CVW_SPS %VBOASG %P 2:A860 = !T7 & !T9, 3: BOASG
         $OUT[860] = NOT $TIMER_FLAG[7] AND NOT $TIMER_FLAG[9]
      ;ENDFOLD
      ;FOLD -- Warte Fraesen fertig oder Timeout -- ;%{SE}%MKUKATPVW %CVW_COM %VCOMMENT %P 2:-- Warte Fraesen fertig oder Timeout --, 3: VW_COMMENT
      ;ENDFOLD
      ;FOLD Schritt 280 = (F79 & F98 + F78 & F94 & !F287 + F78 & F96 & F287 + T7 + T9) & A4039 ;%{SE}%MKUKATPVW %CVW_SPS %VST_CON %P 2:Schritt 280 = (F79 & F98 + F78 & F94 & !F287 + F78 & F96 & F287 + T7 + T9) & A4039, 3: ST_CON
         IF ($FLAG[79] AND $FLAG[98] OR $FLAG[78] AND $FLAG[94] AND NOT $FLAG[287] OR $FLAG[78] AND $FLAG[96] AND $FLAG[287] OR $TIMER_FLAG[7] OR $TIMER_FLAG[9]) AND $OUT[4039] THEN
            PREVSTEP = $APP_INT[5]
            $APP_INT[5] = 280
         ENDIF
      ;ENDFOLD
   ;ENDFOLD
   ;FOLD SCHRITT 280 -- ROB STP1 SZ1 # Ende-- ;%{P}%MKUKATPVW,%CSTEP,%VST_NR,%P 1:SCHRITT, 2:280, 3: ROB STP1 SZ1 # Ende
      ;FOLD ;%{H}
         Case 280
      ;ENDFOLD
      ;FOLD t7 ( EIN ) = STOP ;%{SE}%MKUKATPVW %CVW_SPS %VTSTOP %P 2:t7 ( EIN ) = STOP, 3: TSTOP
         VW(#SET_TIME,TRUE,7,1,0)
      ;ENDFOLD
      ;FOLD -- Wartezeit Programmwechsel SK -- ;%{SE}%MKUKATPVW %CVW_COM %VCOMMENT %P 2:-- Wartezeit Programmwechsel SK --, 3: VW_COMMENT
      ;ENDFOLD
      ;FOLD t8 ( EIN ) = -1[1/10Sek] ;%{SE}%MKUKATPVW %CVW_SPS %VTASG %P 2:t8 ( EIN ) = -1[1/10Sek], 3: TASG
         VW(#SET_TIME,TRUE,8,0,-1)
      ;ENDFOLD
      ;FOLD -- EZ1/SP1/KE1 SZ1 oeffnen -- ;%{SE}%MKUKATPVW %CVW_COM %VCOMMENT %P 2:-- EZ1/SP1/KE1 SZ1 oeffnen --, 3: VW_COMMENT
      ;ENDFOLD
      ;FOLD A718 = AUS ;%{SE}%MKUKATPVW %CVW_SPS %VBOASG %P 2:A718 = AUS, 3: BOASG
         $OUT[718] = FALSE
      ;ENDFOLD
      ;FOLD A717 = EIN ;%{SE}%MKUKATPVW %CVW_SPS %VBOASG %P 2:A717 = EIN, 3: BOASG
         $OUT[717] = TRUE
      ;ENDFOLD
      ;FOLD -- KF1 Ausblasen -- ;%{SE}%MKUKATPVW %CVW_COM %VCOMMENT %P 2:-- KF1 Ausblasen --, 3: VW_COMMENT
      ;ENDFOLD
      ;FOLD A836 = !F298 ;%{SE}%MKUKATPVW %CVW_SPS %VBOASG %P 2:A836 = !F298, 3: BOASG
         $OUT[836] = NOT $FLAG[298]
      ;ENDFOLD
      ;FOLD A860 = A836 & F537 ;%{SE}%MKUKATPVW %CVW_SPS %VBOASG %P 2:A860 = A836 & F537, 3: BOASG
         $OUT[860] = $OUT[836] AND $FLAG[537]
      ;ENDFOLD
      ;FOLD -- RSK Sammelstoerung -- ;%{SE}%MKUKATPVW %CVW_COM %VCOMMENT %P 2:-- RSK Sammelstoerung --, 3: VW_COMMENT
      ;ENDFOLD
      ;FOLD F329 = T7 + T9 ;%{SE}%MKUKATPVW %CVW_SPS %VBOASG %P 2:F329 = T7 + T9, 3: BOASG
         $FLAG[329] = $TIMER_FLAG[7] OR $TIMER_FLAG[9]
      ;ENDFOLD
      ;FOLD -- Hilfsflag Startfraesen -- ;%{SE}%MKUKATPVW %CVW_COM %VCOMMENT %P 2:-- Hilfsflag Startfraesen --, 3: VW_COMMENT
      ;ENDFOLD
      ;FOLD F96 = (F96 & F78 + F98 & F79) & F287 ;%{SE}%MKUKATPVW %CVW_SPS %VBOASG %P 2:F96 = (F96 & F78 + F98 & F79) & F287, 3: BOASG
         $FLAG[96] = ($FLAG[96] AND $FLAG[78] OR $FLAG[98] AND $FLAG[79]) AND $FLAG[287]
      ;ENDFOLD
      ;FOLD F98 = !F130 & F98 + F130 & F287 & F98 ;%{SE}%MKUKATPVW %CVW_SPS %VBOASG %P 2:F98 = !F130 & F98 + F130 & F287 & F98, 3: BOASG
         $FLAG[98] = NOT $FLAG[130] AND $FLAG[98] OR $FLAG[130] AND $FLAG[287] AND $FLAG[98]
      ;ENDFOLD
      ;FOLD F287 = F78 + F79 & F130 ;%{SE}%MKUKATPVW %CVW_SPS %VBOASG %P 2:F287 = F78 + F79 & F130, 3: BOASG
         $FLAG[287] = $FLAG[78] OR $FLAG[79] AND $FLAG[130]
      ;ENDFOLD
      ;FOLD -- Neues Fraesprogramm und Zaehler ruecksetzen -- ;%{SE}%MKUKATPVW %CVW_COM %VCOMMENT %P 2:-- Neues Fraesprogramm und Zaehler ruecksetzen --, 3: VW_COMMENT
      ;ENDFOLD
      ;FOLD bin3 ( F130 ) = 36 ;%{SE}%MKUKATPVW %CVW_SPS %VARIASG %P 2:bin3 ( F130 ) = 36, 3: ARIASG
         VW(#BINOUT,$FLAG[130],3,36)
      ;ENDFOLD
      ;FOLD i4 ( F96 ) = i45 ;%{SE}%MKUKATPVW %CVW_SPS %VARIASG %P 2:i4 ( F96 ) = i45, 3: ARIASG
         VW(#COUNTER,$FLAG[96],4,$COUNT_I[45])
      ;ENDFOLD
      ;FOLD -- Wiederholung beim Startfraesen -- ;%{SE}%MKUKATPVW %CVW_COM %VCOMMENT %P 2:-- Wiederholung beim Startfraesen --, 3: VW_COMMENT
      ;ENDFOLD
      ;FOLD Schritt 276 = E717 & !E718 & (F78 & !F96 + F79 & F130 & !F96) & !F329 & A4039 ;%{SE}%MKUKATPVW %CVW_SPS %VST_CON %P 2:Schritt 276 = E717 & !E718 & (F78 & !F96 + F79 & F130 & !F96) & !F329 & A4039, 3: ST_CON
         IF $IN[717] AND NOT $IN[718] AND ($FLAG[78] AND NOT $FLAG[96] OR $FLAG[79] AND $FLAG[130] AND NOT $FLAG[96]) AND NOT $FLAG[329] AND $OUT[4039] THEN
            PREVSTEP = $APP_INT[5]
            $APP_INT[5] = 276
         ENDIF
      ;ENDFOLD
